PROPERTY ExecuteModelCode_Online : BOOL
GET
hResult := GetObjPara(16#00000008,sizeof(ExecuteModelCode_Online),adr(ExecuteModelCode_Online));
END_GET
SET
hResult := SetObjPara(16#00000008,sizeof(ExecuteModelCode_Online),adr(ExecuteModelCode_Online));
END_SET
END_PROPERTY

PROPERTY ExecuteModelCode_Startup : BOOL
GET
ExecuteModelCode_Startup := stInitData.ExecuteModelCode;
END_GET
SET
stInitData.ExecuteModelCode := ExecuteModelCode_Startup;
END_SET
END_PROPERTY

PROPERTY ExecutionSequence_Online : TctModuleExecutionSequenceType
GET
hResult := GetObjPara(16#00000001,sizeof(ExecutionSequence_Online),adr(ExecutionSequence_Online));
END_GET
SET
hResult := SetObjPara(16#00000001,sizeof(ExecutionSequence_Online),adr(ExecutionSequence_Online));
END_SET
END_PROPERTY

PROPERTY ExecutionSequence_Startup : TctModuleExecutionSequenceType
GET
ExecutionSequence_Startup := stInitData.ExecutionSequence;
END_GET
SET
stInitData.ExecutionSequence := ExecutionSequence_Startup;
END_SET
END_PROPERTY

METHOD FB_init : BOOL
VAR_INPUT
	/// if TRUE, the retain variables are initialized (warm start / cold start)
	bInitRetains: BOOL;
	/// if TRUE, the instance afterwards gets moved into the copy code (online change)
	bInCopyCode: BOOL;
	oid: OTCID;
END_VAR
VAR
	clsId: CLSID;
END_VAR

// initialize flags
bParametersVerified := false;
                    
// set module class id for compatibility check
clsId.Data1 := 16#4ef20903;
clsId.Data2 := 16#d648;
clsId.Data3 := 16#49c7;
clsId.Data4[0] := 16#a9;
clsId.Data4[1] := 16#06;
clsId.Data4[2] := 16#8c;
clsId.Data4[3] := 16#fc;
clsId.Data4[4] := 16#20;
clsId.Data4[5] := 16#50;
clsId.Data4[6] := 16#7f;
clsId.Data4[7] := 16#b3;

AssignClassId(clsId);
                    
// initialize InitData structure with default values              
stInitData.CallByHdr.indexGroup := 0;
stInitData.CallByHdr.indexOffset := 16#00000000;
stInitData.CallByHdr.cbData := SIZEOF(stInitData.CallBy);
stInitData.CallBy := TctModuleCallByType.Module;
stInitData.ExecutionSequenceHdr.indexGroup := 0;
stInitData.ExecutionSequenceHdr.indexOffset := 16#00000001;
stInitData.ExecutionSequenceHdr.cbData := SIZEOF(stInitData.ExecutionSequence);
stInitData.ExecutionSequence := TctModuleExecutionSequenceType.StateUpdateAfterOutputMapping;
stInitData.StepSizeHdr.indexGroup := 0;
stInitData.StepSizeHdr.indexOffset := 16#00000002;
stInitData.StepSizeHdr.cbData := SIZEOF(stInitData.StepSize);
stInitData.StepSize := TctStepSizeType.UseTaskCycleTime;
stInitData.ExecuteModelCodeHdr.indexGroup := 0;
stInitData.ExecuteModelCodeHdr.indexOffset := 16#00000008;
stInitData.ExecuteModelCodeHdr.cbData := SIZEOF(stInitData.ExecuteModelCode);
stInitData.ExecuteModelCode := 1;
stInitData.ModelParametersHdr.indexGroup := 0;
stInitData.ModelParametersHdr.indexOffset := 16#83000000;
stInitData.ModelParametersHdr.cbData := SIZEOF(stInitData.ModelParameters);
stInitData.ModelParameters.DiscreteFilter_NumCoef[0] := 1.25663706143591720e+01;
stInitData.ModelParameters.DiscreteFilter_NumCoef[1] := 1.25663706143591720e+01;
stInitData.ModelParameters.DiscreteFilter_DenCoef[0] := 2.01256637061435910e+03;
stInitData.ModelParameters.DiscreteFilter_DenCoef[1] := -1.98743362938564090e+03;
stInitData.ModelParameters.DiscreteFilter_InitialStates := 0.00000000000000000e+00;
stInitData.ModelParameters.DiscreteFilter1_NumCoef[0] := 1.25663706143591720e+01;
stInitData.ModelParameters.DiscreteFilter1_NumCoef[1] := 1.25663706143591720e+01;
stInitData.ModelParameters.DiscreteFilter1_DenCoef[0] := 2.01256637061435910e+03;
stInitData.ModelParameters.DiscreteFilter1_DenCoef[1] := -1.98743362938564090e+03;
stInitData.ModelParameters.DiscreteFilter1_InitialStates := 0.00000000000000000e+00;
stInitData.ModelParameters.DiscreteFilter2_NumCoef[0] := 1.25663706143591720e+01;
stInitData.ModelParameters.DiscreteFilter2_NumCoef[1] := 1.25663706143591720e+01;
stInitData.ModelParameters.DiscreteFilter2_DenCoef[0] := 2.01256637061435910e+03;
stInitData.ModelParameters.DiscreteFilter2_DenCoef[1] := -1.98743362938564090e+03;
stInitData.ModelParameters.DiscreteFilter2_InitialStates := 0.00000000000000000e+00;
stInitData.ModelParameters.DiscreteFilter3_NumCoef[0] := 1.25663706143591720e+01;
stInitData.ModelParameters.DiscreteFilter3_NumCoef[1] := 1.25663706143591720e+01;
stInitData.ModelParameters.DiscreteFilter3_DenCoef[0] := 2.01256637061435910e+03;
stInitData.ModelParameters.DiscreteFilter3_DenCoef[1] := -1.98743362938564090e+03;
stInitData.ModelParameters.DiscreteFilter3_InitialStates := 0.00000000000000000e+00;
stInitData.ModelParameters.DiscreteFilter4_NumCoef[0] := 1.25663706143591720e+01;
stInitData.ModelParameters.DiscreteFilter4_NumCoef[1] := 1.25663706143591720e+01;
stInitData.ModelParameters.DiscreteFilter4_DenCoef[0] := 2.01256637061435910e+03;
stInitData.ModelParameters.DiscreteFilter4_DenCoef[1] := -1.98743362938564090e+03;
stInitData.ModelParameters.DiscreteFilter4_InitialStates := 0.00000000000000000e+00;
stInitData.ModelParameters.DiscreteFilter5_NumCoef[0] := 1.25663706143591720e+01;
stInitData.ModelParameters.DiscreteFilter5_NumCoef[1] := 1.25663706143591720e+01;
stInitData.ModelParameters.DiscreteFilter5_DenCoef[0] := 2.01256637061435910e+03;
stInitData.ModelParameters.DiscreteFilter5_DenCoef[1] := -1.98743362938564090e+03;
stInitData.ModelParameters.DiscreteFilter5_InitialStates := 0.00000000000000000e+00;
stInitData.ModelParameters.DiscreteFilter6_NumCoef[0] := 1.25663706143591720e+01;
stInitData.ModelParameters.DiscreteFilter6_NumCoef[1] := 1.25663706143591720e+01;
stInitData.ModelParameters.DiscreteFilter6_DenCoef[0] := 2.01256637061435910e+03;
stInitData.ModelParameters.DiscreteFilter6_DenCoef[1] := -1.98743362938564090e+03;
stInitData.ModelParameters.DiscreteFilter6_InitialStates := 0.00000000000000000e+00;
stInitData.ModelParameters.DiscreteFilter7_NumCoef[0] := 1.25663706143591720e+01;
stInitData.ModelParameters.DiscreteFilter7_NumCoef[1] := 1.25663706143591720e+01;
stInitData.ModelParameters.DiscreteFilter7_DenCoef[0] := 2.01256637061435910e+03;
stInitData.ModelParameters.DiscreteFilter7_DenCoef[1] := -1.98743362938564090e+03;
stInitData.ModelParameters.DiscreteFilter7_InitialStates := 0.00000000000000000e+00;
stInitData.ModelParameters.DiscreteFilter8_NumCoef[0] := 1.25663706143591720e+01;
stInitData.ModelParameters.DiscreteFilter8_NumCoef[1] := 1.25663706143591720e+01;
stInitData.ModelParameters.DiscreteFilter8_DenCoef[0] := 2.01256637061435910e+03;
stInitData.ModelParameters.DiscreteFilter8_DenCoef[1] := -1.98743362938564090e+03;
stInitData.ModelParameters.DiscreteFilter8_InitialStates := 0.00000000000000000e+00;
stInitData.ModelParameters.DiscreteFilter9_NumCoef[0] := 1.25663706143591720e+01;
stInitData.ModelParameters.DiscreteFilter9_NumCoef[1] := 1.25663706143591720e+01;
stInitData.ModelParameters.DiscreteFilter9_DenCoef[0] := 2.01256637061435910e+03;
stInitData.ModelParameters.DiscreteFilter9_DenCoef[1] := -1.98743362938564090e+03;
stInitData.ModelParameters.DiscreteFilter9_InitialStates := 0.00000000000000000e+00;
stInitData.ModelParameters.DiscreteFilter10_NumCoef[0] := 1.25663706143591720e+01;
stInitData.ModelParameters.DiscreteFilter10_NumCoef[1] := 1.25663706143591720e+01;
stInitData.ModelParameters.DiscreteFilter10_DenCoef[0] := 2.01256637061435910e+03;
stInitData.ModelParameters.DiscreteFilter10_DenCoef[1] := -1.98743362938564090e+03;
stInitData.ModelParameters.DiscreteFilter10_InitialStates := 0.00000000000000000e+00;
stInitData.ModelParameters.DiscreteFilter11_NumCoef[0] := 1.25663706143591720e+01;
stInitData.ModelParameters.DiscreteFilter11_NumCoef[1] := 1.25663706143591720e+01;
stInitData.ModelParameters.DiscreteFilter11_DenCoef[0] := 2.01256637061435910e+03;
stInitData.ModelParameters.DiscreteFilter11_DenCoef[1] := -1.98743362938564090e+03;
stInitData.ModelParameters.DiscreteFilter11_InitialStates := 0.00000000000000000e+00;
stInitData.ModelParameters.DiscreteFilter12_NumCoef[0] := 1.25663706143591720e+01;
stInitData.ModelParameters.DiscreteFilter12_NumCoef[1] := 1.25663706143591720e+01;
stInitData.ModelParameters.DiscreteFilter12_DenCoef[0] := 2.01256637061435910e+03;
stInitData.ModelParameters.DiscreteFilter12_DenCoef[1] := -1.98743362938564090e+03;
stInitData.ModelParameters.DiscreteFilter12_InitialStates := 0.00000000000000000e+00;
stInitData.ModelParameters.DiscreteFilter13_NumCoef[0] := 1.25663706143591720e+01;
stInitData.ModelParameters.DiscreteFilter13_NumCoef[1] := 1.25663706143591720e+01;
stInitData.ModelParameters.DiscreteFilter13_DenCoef[0] := 2.01256637061435910e+03;
stInitData.ModelParameters.DiscreteFilter13_DenCoef[1] := -1.98743362938564090e+03;
stInitData.ModelParameters.DiscreteFilter13_InitialStates := 0.00000000000000000e+00;
stInitData.ModelParameters.DiscreteFilter14_NumCoef[0] := 1.25663706143591720e+01;
stInitData.ModelParameters.DiscreteFilter14_NumCoef[1] := 1.25663706143591720e+01;
stInitData.ModelParameters.DiscreteFilter14_DenCoef[0] := 2.01256637061435910e+03;
stInitData.ModelParameters.DiscreteFilter14_DenCoef[1] := -1.98743362938564090e+03;
stInitData.ModelParameters.DiscreteFilter14_InitialStates := 0.00000000000000000e+00;
stInitData.ModelParameters.DiscreteFilter15_NumCoef[0] := 1.25663706143591720e+01;
stInitData.ModelParameters.DiscreteFilter15_NumCoef[1] := 1.25663706143591720e+01;
stInitData.ModelParameters.DiscreteFilter15_DenCoef[0] := 2.01256637061435910e+03;
stInitData.ModelParameters.DiscreteFilter15_DenCoef[1] := -1.98743362938564090e+03;
stInitData.ModelParameters.DiscreteFilter15_InitialStates := 0.00000000000000000e+00;
stInitData.ModelParameters.DiscreteFilter16_NumCoef[0] := 1.25663706143591720e+01;
stInitData.ModelParameters.DiscreteFilter16_NumCoef[1] := 1.25663706143591720e+01;
stInitData.ModelParameters.DiscreteFilter16_DenCoef[0] := 2.01256637061435910e+03;
stInitData.ModelParameters.DiscreteFilter16_DenCoef[1] := -1.98743362938564090e+03;
stInitData.ModelParameters.DiscreteFilter16_InitialStates := 0.00000000000000000e+00;
stInitData.ModelParameters.DiscreteFilter17_NumCoef[0] := 1.25663706143591720e+01;
stInitData.ModelParameters.DiscreteFilter17_NumCoef[1] := 1.25663706143591720e+01;
stInitData.ModelParameters.DiscreteFilter17_DenCoef[0] := 2.01256637061435910e+03;
stInitData.ModelParameters.DiscreteFilter17_DenCoef[1] := -1.98743362938564090e+03;
stInitData.ModelParameters.DiscreteFilter17_InitialStates := 0.00000000000000000e+00;
stInitData.ContextInfoArr_0_TaskOidHdr.indexGroup := 0;
stInitData.ContextInfoArr_0_TaskOidHdr.indexOffset := 16#03002060;
stInitData.ContextInfoArr_0_TaskOidHdr.cbData := SIZEOF(stInitData.ContextInfoArr_0_TaskOid);
stInitData.ContextInfoArr_0_TaskPriorityHdr.indexGroup := 0;
stInitData.ContextInfoArr_0_TaskPriorityHdr.indexOffset := 16#03002070;
stInitData.ContextInfoArr_0_TaskPriorityHdr.cbData := SIZEOF(stInitData.ContextInfoArr_0_TaskPriority);
stInitData.ContextInfoArr_0_TaskCycleTimeNsHdr.indexGroup := 0;
stInitData.ContextInfoArr_0_TaskCycleTimeNsHdr.indexOffset := 16#03002080;
stInitData.ContextInfoArr_0_TaskCycleTimeNsHdr.cbData := SIZEOF(stInitData.ContextInfoArr_0_TaskCycleTimeNs);
stInitData.ContextInfoArr_0_TaskPortHdr.indexGroup := 0;
stInitData.ContextInfoArr_0_TaskPortHdr.indexOffset := 16#03002090;
stInitData.ContextInfoArr_0_TaskPortHdr.cbData := SIZEOF(stInitData.ContextInfoArr_0_TaskPort);
stInitData.ContextInfoArr_0_TaskSortOrderHdr.indexGroup := 0;
stInitData.ContextInfoArr_0_TaskSortOrderHdr.indexOffset := 16#030020b0;
stInitData.ContextInfoArr_0_TaskSortOrderHdr.cbData := SIZEOF(stInitData.ContextInfoArr_0_TaskSortOrder);
stInitData.Header.cbData := SIZEOF(stInitData)-SIZEOF(stInitData.Header);
stInitData.Header.uiElmCnt := 10;


// set pointer to InitData structure
SetInitDataInfo(ADR(stInitData));

// set DataArea information
SetDataAreaInfo(ADR(arrDataAreas),2);
arrDataAreas[1].nDataAreaId := 0;
arrDataAreas[1].nSize := SIZEOF(stInput);
arrDataAreas[1].pPlcVar := ADR(stInput);
arrDataAreas[1].pModuleProcImg := 0;
arrDataAreas[1].eDataAreaType := E_TcMatSimDataAreaType.InputDst;
arrDataAreas[2].nDataAreaId := 1;
arrDataAreas[2].nSize := SIZEOF(stOutput);
arrDataAreas[2].pPlcVar := ADR(stOutput);
arrDataAreas[2].pModuleProcImg := 0;
arrDataAreas[2].eDataAreaType := E_TcMatSimDataAreaType.OutputSrc;


// initialize basic interface pointers and return
FB_init := SUCCEEDED(Init(oid));
END_METHOD

PROPERTY InitData : ST_Filter_Current_Hexapod_Robot_InitData
GET
InitData := stInitData;
END_GET
SET
stInitData := InitData;
END_SET
END_PROPERTY

PROPERTY Input_Online : ExtU_Filter_Current_Hexapod_R_T
GET
hResult := GetObjPara(16#80000000,sizeof(Input_Online),adr(Input_Online));
END_GET
SET
hResult := SetObjPara(16#80000000,sizeof(Input_Online),adr(Input_Online));
END_SET
END_PROPERTY

{attribute 'object_name' := 'Internal_SetObjState'}
METHOD PROTECTED Internal_SetObjState
VAR_INPUT
	hr: REFERENCE TO HRESULT;
	nextState: TCOM_STATE;
END_VAR

// update pointer to InitData structure
SetInitDataInfo(ADR(stInitData));
// call base method
SUPER^.Internal_SetObjState(hr,nextState);
END_METHOD

PROPERTY MdlInitialized_Online : BOOL
GET
hResult := GetObjPara(16#00000003,sizeof(MdlInitialized_Online),adr(MdlInitialized_Online));
END_GET
SET
hResult := SetObjPara(16#00000003,sizeof(MdlInitialized_Online),adr(MdlInitialized_Online));
END_SET
END_PROPERTY

PROPERTY ModelParameters_Online : P_Filter_Current_Hexapod_Robo_T
GET
hResult := GetObjPara(16#83000000,sizeof(ModelParameters_Online),adr(ModelParameters_Online));
END_GET
SET
hResult := SetObjPara(16#83000000,sizeof(ModelParameters_Online),adr(ModelParameters_Online));
END_SET
END_PROPERTY

PROPERTY ModelParameters_Startup : P_Filter_Current_Hexapod_Robo_T
GET
ModelParameters_Startup := stInitData.ModelParameters;
END_GET
SET
stInitData.ModelParameters := ModelParameters_Startup;
END_SET
END_PROPERTY

PROPERTY ModuleBuildInfo_Online : TctModuleBuildInfoType
GET
hResult := GetObjPara(16#00000007,sizeof(ModuleBuildInfo_Online),adr(ModuleBuildInfo_Online));
END_GET
SET
hResult := SetObjPara(16#00000007,sizeof(ModuleBuildInfo_Online),adr(ModuleBuildInfo_Online));
END_SET
END_PROPERTY

PROPERTY ModuleInfo_Online : TctModuleInfoType
GET
hResult := GetObjPara(16#00000006,sizeof(ModuleInfo_Online),adr(ModuleInfo_Online));
END_GET
SET
hResult := SetObjPara(16#00000006,sizeof(ModuleInfo_Online),adr(ModuleInfo_Online));
END_SET
END_PROPERTY

{attribute 'object_name' := 'SaveOnlineParametersForInit'}
METHOD SaveOnlineParametersForInit : HRESULT
VAR
	idx: UINT;
	pInitElemHdr: POINTER TO TComInitDataElmHdr;
	pData: PVOID;
	nData: UDINT;
END_VAR
VAR CONSTANT
	nInitDataAlignment: UDINT := 4;
END_VAR

// update pointer to InitData structure
SetInitDataInfo(ADR(stInitData));
// call base method
SaveOnlineParametersForInit := SUPER^.SaveOnlineParametersForInit();
END_METHOD

PROPERTY SimulinkTime_Online : LREAL
GET
hResult := GetObjPara(16#00000005,sizeof(SimulinkTime_Online),adr(SimulinkTime_Online));
END_GET
SET
hResult := SetObjPara(16#00000005,sizeof(SimulinkTime_Online),adr(SimulinkTime_Online));
END_SET
END_PROPERTY

PROPERTY StepSize_Online : TctStepSizeType
GET
hResult := GetObjPara(16#00000002,sizeof(StepSize_Online),adr(StepSize_Online));
END_GET
SET
hResult := SetObjPara(16#00000002,sizeof(StepSize_Online),adr(StepSize_Online));
END_SET
END_PROPERTY

PROPERTY StepSize_Startup : TctStepSizeType
GET
StepSize_Startup := stInitData.StepSize;
END_GET
SET
stInitData.StepSize := StepSize_Startup;
END_SET
END_PROPERTY

{attribute 'object_name' := 'VerifyParameters'}
METHOD PRIVATE VerifyParameters : HRESULT
VAR
	moduleCallByParam: TctModuleCallByType;
END_VAR

IF (bParametersVerified) THEN
  VerifyParameters := Tc2_System.E_HRESULTAdsErr.HRESULT_ADS_NOERROR;
ELSE
  VerifyParameters := GetObjPara(stInitData.CallByHdr.indexOffset,SIZEOF(moduleCallByParam),ADR(moduleCallByParam));
  
  // check the "CallBy" parameter to be set to "Module"
  IF (SUCCEEDED(VerifyParameters) AND (moduleCallByParam <> TctModuleCallByType.Module)) THEN
      VerifyParameters := Tc2_System.E_HRESULTAdsErr.INVALIDPARM;
  END_IF
  
  // set the parameters verified flag
  bParametersVerified := SUCCEEDED(VerifyParameters);
END_IF
END_METHOD

END_FUNCTION_BLOCK

// ---- DUTs/Touch_Signal_Detection/FB_Tough_Signal_Detection_Simple.TcPOU
{attribute 'TcDependOnClassFactory' := 'Tough_Signal_Detection_Simple'}
FUNCTION_BLOCK FB_Tough_Signal_Detection_Simple EXTENDS FB_TcMatSimObject
VAR_INPUT
	stInput: ST_Tough_Signal_Detection_Simple_Input;
END_VAR
VAR_OUTPUT
	stOutput: ST_Tough_Signal_Detection_Simple_Output;
END_VAR
VAR
	stInitData: ST_Tough_Signal_Detection_Simple_InitData;
	arrDataAreas: ARRAY[1..2] OF ST_TcMatSimObjectDataAreaInfo;
	bParametersVerified: BOOL;
END_VAR

PROPERTY CallBy_Online : TctModuleCallByType
GET
hResult := GetObjPara(16#00000000,sizeof(CallBy_Online),adr(CallBy_Online));
END_GET
SET
hResult := SetObjPara(16#00000000,sizeof(CallBy_Online),adr(CallBy_Online));
END_SET
END_PROPERTY

PROPERTY CallBy_Startup : TctModuleCallByType
GET
CallBy_Startup := stInitData.CallBy;
END_GET
SET
stInitData.CallBy := CallBy_Startup;
END_SET
END_PROPERTY

PROPERTY ContextInfoArr_0_TaskCycleTimeNs_Online : UDINT
GET
hResult := GetObjPara(16#03002080,sizeof(ContextInfoArr_0_TaskCycleTimeNs_Online),adr(ContextInfoArr_0_TaskCycleTimeNs_Online));
END_GET
SET
hResult := SetObjPara(16#03002080,sizeof(ContextInfoArr_0_TaskCycleTimeNs_Online),adr(ContextInfoArr_0_TaskCycleTimeNs_Online));
END_SET
END_PROPERTY

PROPERTY ContextInfoArr_0_TaskCycleTimeNs_Startup : UDINT
GET
ContextInfoArr_0_TaskCycleTimeNs_Startup := stInitData.ContextInfoArr_0_TaskCycleTimeNs;
END_GET
SET
stInitData.ContextInfoArr_0_TaskCycleTimeNs := ContextInfoArr_0_TaskCycleTimeNs_Startup;
END_SET
END_PROPERTY

PROPERTY ContextInfoArr_0_TaskOid_Online : OTCID
GET
hResult := GetObjPara(16#03002060,sizeof(ContextInfoArr_0_TaskOid_Online),adr(ContextInfoArr_0_TaskOid_Online));
END_GET
SET
hResult := SetObjPara(16#03002060,sizeof(ContextInfoArr_0_TaskOid_Online),adr(ContextInfoArr_0_TaskOid_Online));
END_SET
END_PROPERTY

PROPERTY ContextInfoArr_0_TaskOid_Startup : OTCID
GET
ContextInfoArr_0_TaskOid_Startup := stInitData.ContextInfoArr_0_TaskOid;
END_GET
SET
stInitData.ContextInfoArr_0_TaskOid := ContextInfoArr_0_TaskOid_Startup;
END_SET
END_PROPERTY

PROPERTY ContextInfoArr_0_TaskPort_Online : UINT
GET
hResult := GetObjPara(16#03002090,sizeof(ContextInfoArr_0_TaskPort_Online),adr(ContextInfoArr_0_TaskPort_Online));
END_GET
SET
hResult := SetObjPara(16#03002090,sizeof(ContextInfoArr_0_TaskPort_Online),adr(ContextInfoArr_0_TaskPort_Online));
END_SET
END_PROPERTY

PROPERTY ContextInfoArr_0_TaskPort_Startup : UINT
GET
ContextInfoArr_0_TaskPort_Startup := stInitData.ContextInfoArr_0_TaskPort;
END_GET
SET
stInitData.ContextInfoArr_0_TaskPort := ContextInfoArr_0_TaskPort_Startup;
END_SET
END_PROPERTY

PROPERTY ContextInfoArr_0_TaskPriority_Online : UDINT
GET
hResult := GetObjPara(16#03002070,sizeof(ContextInfoArr_0_TaskPriority_Online),adr(ContextInfoArr_0_TaskPriority_Online));
END_GET
SET
hResult := SetObjPara(16#03002070,sizeof(ContextInfoArr_0_TaskPriority_Online),adr(ContextInfoArr_0_TaskPriority_Online));
END_SET
END_PROPERTY

PROPERTY ContextInfoArr_0_TaskPriority_Startup : UDINT
GET
ContextInfoArr_0_TaskPriority_Startup := stInitData.ContextInfoArr_0_TaskPriority;
END_GET
SET
stInitData.ContextInfoArr_0_TaskPriority := ContextInfoArr_0_TaskPriority_Startup;
END_SET
END_PROPERTY

PROPERTY ContextInfoArr_0_TaskSortOrder_Online : UDINT
GET
hResult := GetObjPara(16#030020b0,sizeof(ContextInfoArr_0_TaskSortOrder_Online),adr(ContextInfoArr_0_TaskSortOrder_Online));
END_GET
SET
hResult := SetObjPara(16#030020b0,sizeof(ContextInfoArr_0_TaskSortOrder_Online),adr(ContextInfoArr_0_TaskSortOrder_Online));
END_SET
END_PROPERTY

PROPERTY ContextInfoArr_0_TaskSortOrder_Startup : UDINT
GET
ContextInfoArr_0_TaskSortOrder_Startup := stInitData.ContextInfoArr_0_TaskSortOrder;
END_GET
SET
stInitData.ContextInfoArr_0_TaskSortOrder := ContextInfoArr_0_TaskSortOrder_Startup;
END_SET
END_PROPERTY

PROPERTY CycleUpdateExecuted_Online : BOOL
GET
hResult := GetObjPara(16#00000004,sizeof(CycleUpdateExecuted_Online),adr(CycleUpdateExecuted_Online));
END_GET
SET
hResult := SetObjPara(16#00000004,sizeof(CycleUpdateExecuted_Online),adr(CycleUpdateExecuted_Online));
END_SET
END_PROPERTY

METHOD Execute : HRESULT

IF (SUCCEEDED(hResult)) THEN
  hResult := VerifyParameters();
END_IF

	// update DataArea information
SetDataAreaInfo(ADR(arrDataAreas),2);
	
	// call base method
Execute := SUPER^.Execute();
END_METHOD

PROPERTY ExecuteModelCode_Online : BOOL
GET
hResult := GetObjPara(16#00000008,sizeof(ExecuteModelCode_Online),adr(ExecuteModelCode_Online));
END_GET
SET
hResult := SetObjPara(16#00000008,sizeof(ExecuteModelCode_Online),adr(ExecuteModelCode_Online));
END_SET
END_PROPERTY

PROPERTY ExecuteModelCode_Startup : BOOL
GET
ExecuteModelCode_Startup := stInitData.ExecuteModelCode;
END_GET
SET
stInitData.ExecuteModelCode := ExecuteModelCode_Startup;
END_SET
END_PROPERTY

PROPERTY ExecutionSequence_Online : TctModuleExecutionSequenceType
GET
hResult := GetObjPara(16#00000001,sizeof(ExecutionSequence_Online),adr(ExecutionSequence_Online));
END_GET
SET
hResult := SetObjPara(16#00000001,sizeof(ExecutionSequence_Online),adr(ExecutionSequence_Online));
END_SET
END_PROPERTY

PROPERTY ExecutionSequence_Startup : TctModuleExecutionSequenceType
GET
ExecutionSequence_Startup := stInitData.ExecutionSequence;
END_GET
SET
stInitData.ExecutionSequence := ExecutionSequence_Startup;
END_SET
END_PROPERTY

METHOD FB_init : BOOL
VAR_INPUT
	/// if TRUE, the retain variables are initialized (warm start / cold start)
	bInitRetains: BOOL;
	/// if TRUE, the instance afterwards gets moved into the copy code (online change)
	bInCopyCode: BOOL;
	oid: OTCID;
END_VAR
VAR
	clsId: CLSID;
END_VAR

// initialize flags
bParametersVerified := false;
                    
// set module class id for compatibility check
clsId.Data1 := 16#edbb4036;
clsId.Data2 := 16#240d;
clsId.Data3 := 16#4fd3;
clsId.Data4[0] := 16#9b;
clsId.Data4[1] := 16#53;
clsId.Data4[2] := 16#34;
clsId.Data4[3] := 16#bf;
clsId.Data4[4] := 16#ff;
clsId.Data4[5] := 16#27;
clsId.Data4[6] := 16#d6;
clsId.Data4[7] := 16#ef;

AssignClassId(clsId);
                    
// initialize InitData structure with default values              
stInitData.CallByHdr.indexGroup := 0;
stInitData.CallByHdr.indexOffset := 16#00000000;
stInitData.CallByHdr.cbData := SIZEOF(stInitData.CallBy);
stInitData.CallBy := TctModuleCallByType.Module;
stInitData.ExecutionSequenceHdr.indexGroup := 0;
stInitData.ExecutionSequenceHdr.indexOffset := 16#00000001;
stInitData.ExecutionSequenceHdr.cbData := SIZEOF(stInitData.ExecutionSequence);
stInitData.ExecutionSequence := TctModuleExecutionSequenceType.StateUpdateAfterOutputMapping;
stInitData.StepSizeHdr.indexGroup := 0;
stInitData.StepSizeHdr.indexOffset := 16#00000002;
stInitData.StepSizeHdr.cbData := SIZEOF(stInitData.StepSize);
stInitData.StepSize := TctStepSizeType.UseTaskCycleTime;
stInitData.ExecuteModelCodeHdr.indexGroup := 0;
stInitData.ExecuteModelCodeHdr.indexOffset := 16#00000008;
stInitData.ExecuteModelCodeHdr.cbData := SIZEOF(stInitData.ExecuteModelCode);
stInitData.ExecuteModelCode := 1;
stInitData.ModelParametersHdr.indexGroup := 0;
stInitData.ModelParametersHdr.indexOffset := 16#83000000;
stInitData.ModelParametersHdr.cbData := SIZEOF(stInitData.ModelParameters);
stInitData.ModelParameters.VariableTimeDelay_MaxDelay := 1.00000000000000000e+00;
stInitData.ModelParameters.VariableTimeDelay_InitOutput := 0.00000000000000000e+00;
stInitData.ModelParameters.VariableTimeDelay1_MaxDelay := 1.00000000000000000e+00;
stInitData.ModelParameters.VariableTimeDelay1_InitOutput := 0.00000000000000000e+00;
stInitData.ModelParameters.VariableTimeDelay2_MaxDelay := 1.00000000000000000e+00;
stInitData.ModelParameters.VariableTimeDelay2_InitOutput := 0.00000000000000000e+00;
stInitData.ModelParameters.VariableTimeDelay3_MaxDelay := 1.00000000000000000e+00;
stInitData.ModelParameters.VariableTimeDelay3_InitOutput := 0.00000000000000000e+00;
stInitData.ModelParameters.VariableTimeDelay4_MaxDelay := 1.00000000000000000e+00;
stInitData.ModelParameters.VariableTimeDelay4_InitOutput := 0.00000000000000000e+00;
stInitData.ModelParameters.VariableTimeDelay5_MaxDelay := 1.00000000000000000e+00;
stInitData.ModelParameters.VariableTimeDelay5_InitOutput := 0.00000000000000000e+00;
stInitData.ModelParameters.VariableTimeDelay6_MaxDelay := 1.00000000000000000e+00;
stInitData.ModelParameters.VariableTimeDelay6_InitOutput := 0.00000000000000000e+00;
stInitData.ModelParameters.VariableTimeDelay7_MaxDelay := 1.00000000000000000e+00;
stInitData.ModelParameters.VariableTimeDelay7_InitOutput := 0.00000000000000000e+00;
stInitData.ModelParameters.VariableTimeDelay8_MaxDelay := 1.00000000000000000e+00;
stInitData.ModelParameters.VariableTimeDelay8_InitOutput := 0.00000000000000000e+00;
stInitData.ModelParameters.VariableTimeDelay9_MaxDelay := 1.00000000000000000e+00;
stInitData.ModelParameters.VariableTimeDelay9_InitOutput := 0.00000000000000000e+00;
stInitData.ModelParameters.VariableTimeDelay10_MaxDelay := 1.00000000000000000e+00;
stInitData.ModelParameters.VariableTimeDelay10_InitOutput := 0.00000000000000000e+00;
stInitData.ModelParameters.VariableTimeDelay11_MaxDelay := 1.00000000000000000e+00;
stInitData.ModelParameters.VariableTimeDelay11_InitOutput := 0.00000000000000000e+00;
stInitData.ModelParameters.VariableTimeDelay12_MaxDelay := 1.00000000000000000e+00;
stInitData.ModelParameters.VariableTimeDelay12_InitOutput := 0.00000000000000000e+00;
stInitData.ModelParameters.VariableTimeDelay13_MaxDelay := 1.00000000000000000e+00;
stInitData.ModelParameters.VariableTimeDelay13_InitOutput := 0.00000000000000000e+00;
stInitData.ModelParameters.VariableTimeDelay14_MaxDelay := 1.00000000000000000e+00;
stInitData.ModelParameters.VariableTimeDelay14_InitOutput := 0.00000000000000000e+00;
stInitData.ModelParameters.VariableTimeDelay15_MaxDelay := 1.00000000000000000e+00;
stInitData.ModelParameters.VariableTimeDelay15_InitOutput := 0.00000000000000000e+00;
stInitData.ModelParameters.VariableTimeDelay16_MaxDelay := 1.00000000000000000e+00;
stInitData.ModelParameters.VariableTimeDelay16_InitOutput := 0.00000000000000000e+00;
stInitData.ModelParameters.VariableTimeDelay17_MaxDelay := 1.00000000000000000e+00;
stInitData.ModelParameters.VariableTimeDelay17_InitOutput := 0.00000000000000000e+00;
stInitData.ModelParameters.DataStoreMemory5_InitialValue[0] := 1.00000000000000000e+00;
stInitData.ModelParameters.DataStoreMemory5_InitialValue[1] := 3.00000000000000000e+00;
stInitData.ModelParameters.DataStoreMemory5_InitialValue[2] := 5.00000000000000000e+00;
stInitData.ModelParameters.DataStoreMemory6_InitialValue[0] := 2.00000000000000000e+00;
stInitData.ModelParameters.DataStoreMemory6_InitialValue[1] := 4.00000000000000000e+00;
stInitData.ModelParameters.DataStoreMemory6_InitialValue[2] := 6.00000000000000000e+00;
stInitData.ModelParameters.DataStoreMemory4_InitialValue[0] := 1;
stInitData.ModelParameters.DataStoreMemory4_InitialValue[1] := 0;
stInitData.ModelParameters.DataStoreMemory4_InitialValue[2] := 1;
stInitData.ModelParameters.DataStoreMemory4_InitialValue[3] := 0;
stInitData.ModelParameters.DataStoreMemory4_InitialValue[4] := 1;
stInitData.ModelParameters.DataStoreMemory4_InitialValue[5] := 0;
stInitData.ContextInfoArr_0_TaskOidHdr.indexGroup := 0;
stInitData.ContextInfoArr_0_TaskOidHdr.indexOffset := 16#03002060;
stInitData.ContextInfoArr_0_TaskOidHdr.cbData := SIZEOF(stInitData.ContextInfoArr_0_TaskOid);
stInitData.ContextInfoArr_0_TaskPriorityHdr.indexGroup := 0;
stInitData.ContextInfoArr_0_TaskPriorityHdr.indexOffset := 16#03002070;
stInitData.ContextInfoArr_0_TaskPriorityHdr.cbData := SIZEOF(stInitData.ContextInfoArr_0_TaskPriority);
stInitData.ContextInfoArr_0_TaskCycleTimeNsHdr.indexGroup := 0;
stInitData.ContextInfoArr_0_TaskCycleTimeNsHdr.indexOffset := 16#03002080;
stInitData.ContextInfoArr_0_TaskCycleTimeNsHdr.cbData := SIZEOF(stInitData.ContextInfoArr_0_TaskCycleTimeNs);
stInitData.ContextInfoArr_0_TaskPortHdr.indexGroup := 0;
stInitData.ContextInfoArr_0_TaskPortHdr.indexOffset := 16#03002090;
stInitData.ContextInfoArr_0_TaskPortHdr.cbData := SIZEOF(stInitData.ContextInfoArr_0_TaskPort);
stInitData.ContextInfoArr_0_TaskSortOrderHdr.indexGroup := 0;
stInitData.ContextInfoArr_0_TaskSortOrderHdr.indexOffset := 16#030020b0;
stInitData.ContextInfoArr_0_TaskSortOrderHdr.cbData := SIZEOF(stInitData.ContextInfoArr_0_TaskSortOrder);
stInitData.Header.cbData := SIZEOF(stInitData)-SIZEOF(stInitData.Header);
stInitData.Header.uiElmCnt := 10;


// set pointer to InitData structure
SetInitDataInfo(ADR(stInitData));

// set DataArea information
SetDataAreaInfo(ADR(arrDataAreas),2);
arrDataAreas[1].nDataAreaId := 0;
arrDataAreas[1].nSize := SIZEOF(stInput);
arrDataAreas[1].pPlcVar := ADR(stInput);
arrDataAreas[1].pModuleProcImg := 0;
arrDataAreas[1].eDataAreaType := E_TcMatSimDataAreaType.InputDst;
arrDataAreas[2].nDataAreaId := 1;
arrDataAreas[2].nSize := SIZEOF(stOutput);
arrDataAreas[2].pPlcVar := ADR(stOutput);
arrDataAreas[2].pModuleProcImg := 0;
arrDataAreas[2].eDataAreaType := E_TcMatSimDataAreaType.OutputSrc;


// initialize basic interface pointers and return
FB_init := SUCCEEDED(Init(oid));
END_METHOD

PROPERTY InitData : ST_Tough_Signal_Detection_Simple_InitData
GET
InitData := stInitData;
END_GET
SET
stInitData := InitData;
END_SET
END_PROPERTY

PROPERTY Input_Online : ExtU_Touch_Signal_Detection_S_T
GET
hResult := GetObjPara(16#80000000,sizeof(Input_Online),adr(Input_Online));
END_GET
SET
hResult := SetObjPara(16#80000000,sizeof(Input_Online),adr(Input_Online));
END_SET
END_PROPERTY

{attribute 'object_name' := 'Internal_SetObjState'}
METHOD PROTECTED Internal_SetObjState
VAR_INPUT
	hr: REFERENCE TO HRESULT;
	nextState: TCOM_STATE;
END_VAR

// update pointer to InitData structure
SetInitDataInfo(ADR(stInitData));
// call base method
SUPER^.Internal_SetObjState(hr,nextState);
END_METHOD

PROPERTY MdlInitialized_Online : BOOL
GET
hResult := GetObjPara(16#00000003,sizeof(MdlInitialized_Online),adr(MdlInitialized_Online));
END_GET
SET
hResult := SetObjPara(16#00000003,sizeof(MdlInitialized_Online),adr(MdlInitialized_Online));
END_SET
END_PROPERTY

PROPERTY ModelParameters_Online : P_Touch_Signal_Detection_Simp_T
GET
hResult := GetObjPara(16#83000000,sizeof(ModelParameters_Online),adr(ModelParameters_Online));
END_GET
SET
hResult := SetObjPara(16#83000000,sizeof(ModelParameters_Online),adr(ModelParameters_Online));
END_SET
END_PROPERTY

PROPERTY ModelParameters_Startup : P_Touch_Signal_Detection_Simp_T
GET
ModelParameters_Startup := stInitData.ModelParameters;
END_GET
SET
stInitData.ModelParameters := ModelParameters_Startup;
END_SET
END_PROPERTY

PROPERTY ModuleBuildInfo_Online : TctModuleBuildInfoType
GET
hResult := GetObjPara(16#00000007,sizeof(ModuleBuildInfo_Online),adr(ModuleBuildInfo_Online));
END_GET
SET
hResult := SetObjPara(16#00000007,sizeof(ModuleBuildInfo_Online),adr(ModuleBuildInfo_Online));
END_SET
END_PROPERTY

PROPERTY ModuleInfo_Online : TctModuleInfoType
GET
hResult := GetObjPara(16#00000006,sizeof(ModuleInfo_Online),adr(ModuleInfo_Online));
END_GET
SET
hResult := SetObjPara(16#00000006,sizeof(ModuleInfo_Online),adr(ModuleInfo_Online));
END_SET
END_PROPERTY

{attribute 'object_name' := 'SaveOnlineParametersForInit'}
METHOD SaveOnlineParametersForInit : HRESULT
VAR
	idx: UINT;
	pInitElemHdr: POINTER TO TComInitDataElmHdr;
	pData: PVOID;
	nData: UDINT;
END_VAR
VAR CONSTANT
	nInitDataAlignment: UDINT := 4;
END_VAR

// update pointer to InitData structure
SetInitDataInfo(ADR(stInitData));
// call base method
SaveOnlineParametersForInit := SUPER^.SaveOnlineParametersForInit();
END_METHOD

PROPERTY SimulinkTime_Online : LREAL
GET
hResult := GetObjPara(16#00000005,sizeof(SimulinkTime_Online),adr(SimulinkTime_Online));
END_GET
SET
hResult := SetObjPara(16#00000005,sizeof(SimulinkTime_Online),adr(SimulinkTime_Online));
END_SET
END_PROPERTY

PROPERTY StepSize_Online : TctStepSizeType
GET
hResult := GetObjPara(16#00000002,sizeof(StepSize_Online),adr(StepSize_Online));
END_GET
SET
hResult := SetObjPara(16#00000002,sizeof(StepSize_Online),adr(StepSize_Online));
END_SET
END_PROPERTY

PROPERTY StepSize_Startup : TctStepSizeType
GET
StepSize_Startup := stInitData.StepSize;
END_GET
SET
stInitData.StepSize := StepSize_Startup;
END_SET
END_PROPERTY

{attribute 'object_name' := 'VerifyParameters'}
METHOD PRIVATE VerifyParameters : HRESULT
VAR
	moduleCallByParam: TctModuleCallByType;
END_VAR

IF (bParametersVerified) THEN
  VerifyParameters := Tc2_System.E_HRESULTAdsErr.HRESULT_ADS_NOERROR;
ELSE
  VerifyParameters := GetObjPara(stInitData.CallByHdr.indexOffset,SIZEOF(moduleCallByParam),ADR(moduleCallByParam));
  
  // check the "CallBy" parameter to be set to "Module"
  IF (SUCCEEDED(VerifyParameters) AND (moduleCallByParam <> TctModuleCallByType.Module)) THEN
      VerifyParameters := Tc2_System.E_HRESULTAdsErr.INVALIDPARM;
  END_IF
  
  // set the parameters verified flag
  bParametersVerified := SUCCEEDED(VerifyParameters);
END_IF
END_METHOD

END_FUNCTION_BLOCK

// ---- POUs/Walking_Welding_Robot_Control.TcPOU
PROGRAM Walking_Welding_Robot_Control
VAR_INPUT
	// ====== 整体界面激活 ======
	Walking_Welding_Robot_Joint_Control	: BOOL;				// 允许对界面进行操作,对应UI中的Enable_All_Buttons
	
	// ====== 模块使能信号 ======
	Walking_Welding_Robot_Power 		: BOOL;				// [24电机上电]
	Walking_Welding_Robot_Home_Execute	: BOOL;				// [找零使能]
	Walking_Welding_Robot_Moving_Execute: BOOL;				// [运动使能]
	
	// ====== 控制类型选择 ======
	User_Moving_Control					: BOOL;				// 用户输入目标位置进行运动
	Auto_Moving_Control					: BOOL;				// 机器人自主根据Walking_Robot_Movement的默认参数进行运动
END_VAR

VAR
	// ===================控制信号输入=============
	// 六足运动位置定义(按潘阳坐标系) - 用户操作控制
		// 用户指定目标位置
	Robot_Walking_Z						: LREAL := 1.00;	// 用户指定运动 : Z方向目标位置
	Robot_Walking_X						: LREAL := 0.40;	// 用户指定运动 : X方向目标位置
	Robot_Walking_alpha					: LREAL := pi/12;	// 用户指定运动 : 绕Y轴旋转角度
	Robot_Walking_Velocity				: LREAL := 0.03;	// 用户指定运动 : 机器人运动速度默认0.03m/s
		// 机器人各方向运动速度
	Robot_Walking_Vx					: LREAL;			// X方向运动速度
	Robot_Walking_Vz					: LREAL;			// Z方向运动速度
	Robot_Walking_Va					: LREAL;			// Y方向转动速度
		// 机器人从当前位置运动到目标位置所需时间
	Robot_Walking_t						: LREAL;			// 运动总时间
END_VAR


Logic_Control();			// 逻辑控制程序

Input_Calculate();			// 用户输入参数计算

ACTION Input_Calculate:



// 用户指定目标位置,以当前位置为[0,0,0,0,0,0],按照机器人进行匀速运动,计算三个方向的速度
	// 沿X方向移动的速度分量 Vx = V * sin(theta)
Robot_Walking_Vx 	:= Robot_Walking_Velocity * SIN(ATAN(Robot_Walking_X/Robot_Walking_Z));
	// 沿Z方向移动的速度分量 Vz = V * cos(theta)
Robot_Walking_Vz 	:= Robot_Walking_Velocity * COS(ATAN(Robot_Walking_X/Robot_Walking_Z));
	// 机器人运动的总时间 t = Z / Vz
Robot_Walking_t		:= Robot_Walking_Z / Robot_Walking_Vz;	
	// 沿Y方向转动的速度分量 Va = alpha / t
Robot_Walking_Va	:= Robot_Walking_alpha / Robot_Walking_t;


// Simulink里的模型是以最开始的位置为全局坐标系,走到目标位置后
// 再想走一段的话重新给Vx,Vz,Va会发生什么呢？  

// 如果此时将Simulink模型的输入时间改为t=0会发生什么
END_ACTION

ACTION Logic_Control:
// ************************整体移动焊接机器人控制逻辑***********************

//  激活整个模块后,允许使用界面上的按钮进行操作,这样才能进行整体上电、找零、运动
IF Walking_Welding_Robot_Joint_control THEN
	// 上电、找零、运动三者逻辑
		// 未上电,不能找零和运动
	IF NOT Walking_Welding_Robot_Power THEN
		Walking_Welding_Robot_Home_Execute 	:= FALSE;
		Walking_Welding_Robot_Moving_Execute:= FALSE;
	END_IF
		// 找零时,不能运动
	IF Walking_Welding_Robot_Home_Execute THEN
		Walking_Welding_Robot_Moving_Execute:= FALSE;
	END_IF
		// 运动时,不能找零
	IF Walking_Welding_Robot_Moving_Execute THEN
		Walking_Welding_Robot_Home_Execute 	:= FALSE;
	END_IF	

	// 上电逻辑
		// [24电机上电]开启,则通过对应的控制PRG直接将所有电机整体上电
	IF Walking_Welding_Robot_Power THEN
		Walking_Robot_Control.Power_Execute 	:= TRUE;
		Walking_Robot_Control.Robot_Power		:= TRUE;
		Welding_Arm_Control.Power_Execute 		:= TRUE;
		Welding_Arm_Control.Welding_Arm_Power 	:= TRUE;
		// [24电机上电]关闭,通过对应的控制PRG直接将所有电机整体断电
	ELSIF NOT Walking_Welding_Robot_Power THEN
		Walking_Robot_Control.Power_Execute 	:= FALSE;
		Walking_Robot_Control.Robot_Power		:= FALSE;
		Welding_Arm_Control.Power_Execute 		:= FALSE;	
		Welding_Arm_Control.Welding_Arm_Power	:= FALSE;
	END_IF
		
	// 找零逻辑
		// [找零使能],则允许用户对焊接臂/步行机器人分别进行整体找零
		// 但仅仅是允许,找零动作的发生还需要用户通过界面上的按钮进行操作
	IF Walking_Welding_Robot_Home_Execute THEN
		Walking_Robot_Control.Home_Execute 		:= TRUE;	// 六足找零使能开启
		Walking_Robot_Control.Robot_Home_Set	:= TRUE;	// 六足单组退找零使能开启
		Welding_Arm_Control.Home_Execute 		:= TRUE;	// 焊接臂找零使能开启
	ELSIF NOT Walking_Welding_Robot_Home_Execute THEN
		Walking_Robot_Control.Home_Execute 		:= FALSE;
		Walking_Robot_Control.Robot_Home_Set	:= FALSE;
		Welding_Arm_Control.Home_Execute 		:= FALSE;
	END_IF
	
	// 两种控制方式互斥
	IF User_Moving_Control THEN
		Auto_Moving_Control := FALSE;
	END_IF
	IF Auto_Moving_Control THEN
		User_Moving_Control := FALSE;
	END_IF
	
	// 运动控制逻辑
	IF Walking_Welding_Robot_Moving_Execute THEN
		// [运动使能],则允许用户对焊接臂/步行机器人分别进行运动控制,即两者外部发生使能
		Walking_Robot_Movement.ExSetPoint_Execute 		:= TRUE;
		Welding_Arm_Movement.ExSetPoint_Execute 		:= TRUE;

		IF User_Moving_Control THEN
			Walking_Robot_Movement.ExtSetPointEnable	:= TRUE;
			Walking_Robot_Movement.ExtSetPointDisable	:= FALSE;
		ELSIF NOT User_Moving_Control THEN
			Walking_Robot_Movement.ExtSetPointEnable	:= FALSE;
			Walking_Robot_Movement.ExtSetPointDisable	:= TRUE;
		END_IF
		
	ELSIF NOT Walking_Welding_Robot_Moving_Execute THEN
		// [运动使能]关闭,不允许控制,且外部发生使能关闭
		Auto_Moving_Control := FALSE;
		User_Moving_Control := FALSE;
		Walking_Robot_Movement.ExSetPoint_Execute 	:= FALSE;
		Welding_Arm_Movement.ExSetPoint_Execute 	:= FALSE;
	END_IF
	
		// 用户自定义行走,走到目标位置后停止
	IF User_Moving_Control THEN
		// 到达目标位置附近后停止
		
		IF (Robot_Walking_Z-Walking_Robot_Movement.Act_Slice[3])< 0.15 AND (Robot_Walking_X-Walking_Robot_Movement.Act_Slice[4])<0.15 THEN
			// 到达目标位置,并且是六条腿支撑(state=2,realstate=3)的情况下,停止运动,并将User_Moving_Control复位
			IF Walking_Robot_Movement.state = 2 AND Walking_Robot_Movement.realState = 3 THEN
				// 先关使能信号,后关Enable和Disable两个外部运动开始信号
				User_Moving_Control := FALSE;
				Walking_Robot_Movement.ExtSetPointEnable 	:= FALSE;
				Walking_Robot_Movement.ExtSetPointDisable	:= TRUE;
			END_IF
		//ELSE
			//Walking_Robot_Movement.ExtSetPointEnable 		:= TRUE;
		END_IF
		
	END_IF
	
	
	// 不激活界面,因此界面所有的按钮默认关闭
ELSIF NOT Walking_Welding_Robot_Joint_Control THEN
	Walking_Welding_Robot_Power 			:= FALSE;
	Walking_Welding_Robot_Home_Execute 		:= FALSE;
	Walking_Welding_Robot_Moving_Execute	:= FALSE;
	User_Moving_Control						:= FALSE;
	Auto_Moving_Control						:= FALSE;
END_IF
END_ACTION

ACTION Variable_Monitor:
// =====================关键数据信号监测======================
END_ACTION

ACTION Variable_Set:

END_ACTION

END_PROGRAM

// ---- POUs/Welding_Arm_Control.TcPOU
PROGRAM Welding_Arm_Control

VAR CONSTANT
	MotorNum					: INT := 6;								// 接入控制的电机数量
END_VAR

VAR_INPUT
	// ====== 模块动作信号(按动作先后排列) ======
	Power_Execute 				: BOOL;									// 上电使能
	Axis_Power					: ARRAY[1..MotorNum] OF BOOL;			// 单电机上电
	Welding_Arm_Power			: BOOL;									// 焊接臂所有电机上电
	
	Home_Execute				: BOOL;									// 找零使能
	Axis_Home_Set				: ARRAY[1..MotorNum] OF BOOL;			// 单电机找零
	Welding_Arm_Home_Set		: BOOL;									// 焊接臂所有电机找零

	Reset_Execute				: BOOL;									// 电机驱动重置使能
	Axis_Reset					: ARRAY[1..MotorNum] OF BOOL;			// 单电机驱动重置
	Welding_Arm_Reset			: BOOL;									// 焊接臂整体电机驱动重置
	
	Welding_Arm_Move_Execute	: BOOL;									// 焊接臂运动程序使能	
	Move_Absolute_Execute		: BOOL;									// 绝对运动使能
	Move_Relative_Execute		: BOOL;									// 相对运动使能
	Axis_Absolute_Eable			: ARRAY[1..MotorNum] OF BOOL;			// 单电机绝对运动使能
	Axis_Relative_Eable			: ARRAY[1..MotorNum] OF BOOL;			// 单电机相对运动使能
	Axis_Move_Absolute_Position	: ARRAY[1..MotorNum] OF LREAL;			// 单电机绝对运动位置
	Axis_Move_Relative_Position	: ARRAY[1..MotorNum] OF LREAL;			// 单电机相对运动位置			
	
END_VAR
VAR
	// ====== NC轴变量 ======
	Axis_Welding_Arm			: ARRAY[1..MotorNum] OF Axis;			// 定义焊接臂轴参量(可以调整数据上限来调整电机数目)
	Axis_Number 				: INT;									// 定义轴数目
	
	// ====== 状态监测变量 ======
	Power_Status				: ARRAY[1..MotorNum] OF BOOL;			// 单电机上电状态
	Home_Done					: ARRAY[1..MotorNum] OF BOOL;			// 单电机找零状态
	Welding_Arm_Home_Done		: BOOL;									// 机器臂找零完成状态
	MoveAbsoluteDone			: ARRAY[1..MotorNum] OF BOOL;			// 单电机绝对运动状态
	MoveRelativeDone			: ARRAY[1..MotorNum] OF BOOL;			// 单电机相对运动状态
	
	Welding_Arm_Error			: BOOL;									// 焊接臂电机错误信号
	Axis_Error					: ARRAY[1..MotorNum] OF BOOL;			// 单电机错误信号
	Axis_ErrorID				: ARRAY[1..MotorNum] OF UDINT;			// 单电机错误码
	
	Axis_ActPostion				: ARRAY[1..MotorNum] OF LREAL;			// 单电机实际位置
	Axis_ActVelocity			: ARRAY[1..MotorNum] OF LREAL;			// 单电机实际速度
	
	Current_Turque_Value  AT%IW0: ARRAY[1..MotorNum] OF INT ;			// 单电机实际电流
	Digital_Inputs  	  AT%I* : ARRAY[1..MotorNum] OF DINT ;			// 驱动数字输入信号（Link到驱动器中的Digital Inputs）
	
	Home_Switch_value 			: ARRAY[1..MotorNum] OF BOOL;			// 限位开关值
	
	Max_Turque_Value 			: INT ;									// 最大电流边界值(机械限位法找零时用来判断运动极限位置)
END_VAR


Variable_Monitor();					// 变量监测程序

Logic_Control();					// 逻辑控制程序

Variable_Set();						// 变量设置程序

Welding_Arm_Action();				// 焊接臂整体运动程序

Welding_Arm_Single_Motor_Action();	// 焊接臂单电机运动程序

//Safety();							// 强安全措施程序

ACTION Logic_Control:
// =======================控制逻辑区==========================
// 保证所有的动作拥有合理的先后顺序，优化控制逻辑
// 也防止出现两个或两个以上动作同时进行的情况，保证控制安全

// ====== 电机驱动重置逻辑 ======
FOR Axis_Number := 1 TO MotorNum {BY 1} DO
	IF Axis_Error[Axis_Number] THEN
		Welding_Arm_Error := TRUE;
		EXIT;
	END_IF
	Welding_Arm_Error := FALSE;
END_FOR

IF Welding_Arm_Error THEN
	Reset_Execute := TRUE;
ELSIF NOT Welding_Arm_Error THEN
	Reset_Execute := FALSE;
END_IF

IF NOT Reset_Execute THEN
	FOR Axis_Number := 1 TO MotorNum {BY 1} DO
		Axis_Reset[Axis_Number] := FALSE;
		Axis_Welding_Arm[Axis_Number].Reset(Drive_Reset:= Axis_Reset[Axis_Number]);
	END_FOR
END_IF
	// 没有错误则不允许按按钮,或清除了错误按钮回弹
FOR Axis_Number := 1 TO MotorNum {BY 1} DO
	IF NOT Axis_Error[Axis_Number] THEN
		Axis_Reset[Axis_Number] := FALSE;
	END_IF
END_FOR

// ====== 上电逻辑 ======
IF NOT Power_Execute THEN
	FOR Axis_Number := 1 TO MotorNum {BY 1} DO
		Axis_Power[Axis_Number] := FALSE;
		Axis_Welding_Arm[Axis_Number].Power(Axis_Enable:= Axis_Power[Axis_Number]);
	END_FOR
END_IF

// ====== 找零逻辑 ======
IF Home_Execute THEN
	FOR Axis_Number := 1 TO MotorNum {BY 1} DO
		IF Home_Done[Axis_Number] THEN			// 	丝杠到达零点位置后，单电机标零使能位关闭			
			Axis_Home_Set[Axis_Number] := FALSE;	
			Axis_Welding_Arm[Axis_Number].Home_Sensor_Backward(	Drive_Home:= Axis_Home_Set[Axis_Number], 
													Home_Switch := NOT Home_Switch_value[Axis_Number]);
		END_IF
	END_FOR
	Move_Absolute_Execute := FALSE;							// 设定零点时，不能进行其他运动
	//ExSetPoint_Execute :=0;
ELSIF NOT Home_Execute THEN
	FOR Axis_Number := 1 TO MotorNum {BY 1} DO
		//Axis_Start_Back[Axis_Number] :=0;
		Axis_Home_Set[Axis_Number] := FALSE;
	END_FOR
END_IF

// ====== 绝对运动逻辑 ======
IF Move_Absolute_Execute THEN
	//Absolute_Eable := TRUE;
	Home_Execute := FALSE;							// 运动运动使能时，焊接臂调零必须结束
	//ExSetPoint_Execute :=0;						// 运动运动时，不能进行其他运动
	FOR Axis_Number := 1 TO MotorNum {BY 1} DO
		IF MoveAbsoluteDone[Axis_Number] THEN		// 	丝杠到达设定位置后，单电机绝对运动使能位关闭
			Axis_Absolute_Eable[Axis_Number] := FALSE;
		END_IF
	END_FOR
ELSIF NOT Move_Absolute_Execute THEN							// 运动不使能,轴不能运动
	FOR Axis_Number := 1 TO MotorNum {BY 1} DO
		Axis_Absolute_Eable[Axis_Number] := FALSE;
		Axis_Welding_Arm[Axis_Number].Move_Absolute(  Drive_Move_Absolute:= Axis_Absolute_Eable[Axis_Number], 
													  Absolute_Position:= Axis_Move_Absolute_Position[Axis_Number]);
	END_FOR
END_IF

// ====== 焊接臂相对运动逻辑 ======
IF Move_Relative_Execute THEN
	//Relative_Eable := TRUE;
	Home_Execute := FALSE;							// 运动运动使能时，焊接臂调零必须结束
	//ExSetPoint_Execute :=0;						// 运动运动时，不能进行其他运动
	FOR Axis_Number := 1 TO MotorNum {BY 1} DO
		IF MoveRelativeDone[Axis_Number] THEN		// 	丝杠到达设定位置后，单电机相对运动使能位关闭
			Axis_Relative_Eable[Axis_Number] := FALSE;
			Axis_Welding_Arm[Axis_Number].Move_Relative(  Drive_Move_Relative:= Axis_Relative_Eable[Axis_Number], 
													  Relative_Position:= Axis_Move_Relative_Position[Axis_Number]);
		END_IF
	END_FOR
ELSIF NOT Move_Relative_Execute THEN							// 运动不使能,轴不能运动
	FOR Axis_Number := 1 TO MotorNum {BY 1} DO
		Axis_Relative_Eable[Axis_Number] := FALSE;
		Axis_Welding_Arm[Axis_Number].Move_Relative(  Drive_Move_Relative:= Axis_Relative_Eable[Axis_Number], 
													  Relative_Position:= Axis_Move_Relative_Position[Axis_Number]);
	END_FOR
END_IF
END_ACTION

ACTION Safety:
// 保证丝杠行程和电机速度在规定范围内

// 如果没在找零，检测到焊接臂升降或径向关节接近开关信号即停止焊接臂上所有电机
IF NOT Home_Execute THEN
	// Digital_Inputs[1].19 为焊接臂升降电机接近开关(下)标识位
	// Digital_Inputs[3].20 为焊接臂径向电机接近开关(远离电机侧)标识位
	IF Digital_Inputs[1].18 OR Digital_Inputs[1].19 OR Digital_Inputs[3].20 OR Digital_Inputs[3].21 THEN
		FOR Axis_Number := 1 TO MotorNum {BY 1} DO
			//Axis_Power[Axis_Number] := FALSE;
		END_FOR
	END_IF
END_IF

//IF Digital_Inputs[1].18 THEN
//	pos_up := Axis_Welding_Arm[1].ActPosition;
//	range_v := pos_down - pos_up;
//	Axis_Power[1] := FALSE;
//END_IF
//IF Digital_Inputs[1].19 THEN
//	pos_down := Axis_Welding_Arm[1].ActPosition;
//	Axis_Move_Relative_Position[1] := -300;
//ELSE
//	Axis_Move_Relative_Position[1] := 200;
//END_IF

//IF Digital_Inputs[2].20 THEN
//	pos_far := Axis_Welding_Arm[2].ActPosition;
//	range_h := pos_far - pos_near;
//	Axis_Power[2] := FALSE;
//END_IF
//IF Digital_Inputs[2].21 THEN
//	pos_near := Axis_Welding_Arm[2].ActPosition;

//	Axis_Move_Relative_Position[2] := 200;
//ELSE
//	Axis_Move_Relative_Position[2] := 3;
//END_IF
END_ACTION

ACTION Variable_Monitor:
// =====================关键数据信号监测======================

// ====== 设置最大力矩(边界控制条件) ======
FOR Axis_Number := 1 TO MotorNum {BY 1} DO
	Axis_Welding_Arm[Axis_Number].Max_Turque_Value := Max_Turque_Value;
END_FOR

// ====== 检测实际力矩 ======
FOR Axis_Number := 1 TO MotorNum {BY 1} DO
	Axis_Welding_Arm[Axis_Number].Current_Turque_Value := Current_Turque_Value[Axis_Number];
END_FOR

// ====== 检测轴实际位置、速度 ======
FOR Axis_Number := 1 TO MotorNum {BY 1} DO
	Axis_ActPostion[Axis_Number] 	:= Axis_Welding_Arm[Axis_Number].ActPosition;
	Axis_ActVelocity[Axis_Number] 	:= Axis_Welding_Arm[Axis_Number].ActVelocity;
END_FOR

// ====== 检测上电状态 ======
FOR Axis_Number := 1 TO MotorNum {BY 1} DO
	Power_Status[Axis_Number] := Axis_Welding_Arm[Axis_Number].State_PowerStatus;
END_FOR

// ====== 检测找零状态 ======
FOR Axis_Number := 1 TO MotorNum {BY 1} DO
	Home_Done[Axis_Number] := Axis_Welding_Arm[Axis_Number].State_HomeDone;
END_FOR

// ====== 检测电机绝对运动状态 ======
FOR Axis_Number := 1 TO MotorNum {BY 1} DO
	MoveAbsoluteDone[Axis_Number] := Axis_Welding_Arm[Axis_Number].State_MoveAbsoluteDone;
END_FOR

// ====== 检测电机相对运动状态 ======
FOR Axis_Number := 1 TO MotorNum {BY 1} DO
	MoveRelativeDone[Axis_Number] := Axis_Welding_Arm[Axis_Number].State_MoveRelativeDone;
END_FOR

// ====== 检测电机错误 ======
FOR Axis_Number := 1 TO MotorNum {BY 1} DO
	Axis_Error[Axis_Number] 	:= Axis_Welding_Arm[Axis_Number].Axis_Error;
	Axis_ErrorID[Axis_Number] 	:= Axis_Welding_Arm[Axis_Number].Axis_ErrorID;
END_FOR
END_ACTION

ACTION Variable_Set:
// ====== 设置速度 ======
FOR Axis_Number := 1 TO MotorNum {BY 1} DO							//此时每一个电机的速度都是一样的
	Axis_Welding_Arm[Axis_Number].Home_Velocity 	:= 5;			//找零速度(Axis_Jog中的速度)
	Axis_Welding_Arm[Axis_Number].Move_Relative_Velocity	:=5;	//相对运动速度
END_FOR
IF Home_Execute THEN
	FOR Axis_Number := 1 TO MotorNum {BY 1} DO
		Axis_Welding_Arm[Axis_Number].Move_Absolute_Velocity := 5;	//找零之后运动至轨迹起始点的速度
	END_FOR
ELSE
	FOR Axis_Number := 1 TO MotorNum {BY 1} DO
			Axis_Welding_Arm[Axis_Number].Move_Absolute_Velocity	:=10;
	END_FOR
END_IF
	

// ====== 设置绝对运动位置 ======
FOR Axis_Number := 1 TO MotorNum {BY 1} DO
	Axis_Move_Absolute_Position[Axis_Number] := 100;
END_FOR

// ====== 设置相对运动距离 ======
FOR Axis_Number := 1 TO MotorNum {BY 1} DO
	Axis_Move_Relative_Position[Axis_Number] := -15;
END_FOR

// ====== 设置最大力矩(找零过程判断已到丝杠顶点) ======
Max_Turque_Value := 1400;

// ====== 设置电机设零后到达Simulink模型初始位置 ======
IF Home_Execute THEN
	FOR Axis_Number := 1 TO MotorNum {BY 1} DO
		Axis_Welding_Arm[Axis_Number].Home_Absolute_Position := Welding_Arm_Movement.ExSetPoint_Position[Axis_Number];
	END_FOR
END_IF
END_ACTION

ACTION Welding_Arm_Action:
// =================焊接臂整体运动命令区======================
// 六足所有电机整体控制

// ====== 焊接臂所有电机驱动重置 ======
IF Welding_Arm_Reset THEN							// 缺少输入
	IF Reset_Execute THEN
		FOR Axis_Number := 1 TO MotorNum {BY 1} DO
			Axis_Reset[Axis_Number] := TRUE;
			Axis_Welding_Arm[Axis_Number].Reset(Drive_Reset:= Axis_Reset[Axis_Number]);
		END_FOR
	END_IF
END_IF	

// ====== 焊接臂所有电机上电 ======
IF Welding_Arm_Power THEN	
	IF Power_Execute THEN
		FOR Axis_Number := 1 TO MotorNum {BY 1} DO
			Axis_Power[Axis_Number] := TRUE ;
		END_FOR
	END_IF
END_IF
	
// ====== 焊接臂所有电机找零 ======
IF Welding_Arm_Home_Set THEN
	IF Home_Execute THEN
		FOR Axis_Number := 1 TO MotorNum {BY 1} DO
			IF NOT Home_Done[Axis_Number] THEN
				Axis_Home_Set[Axis_Number] := TRUE;
				Axis_Welding_Arm[Axis_Number].Home_Sensor_Backward(	Drive_Home:= Axis_Home_Set[Axis_Number], 
													Home_Switch := NOT Home_Switch_value[Axis_Number]);
			ELSIF Home_Done[Axis_Number] THEN
				Axis_Home_Set[Axis_Number] := FALSE;
				Axis_Welding_Arm[Axis_Number].Home_Sensor_Backward(	Drive_Home:= Axis_Home_Set[Axis_Number], 
													Home_Switch := NOT Home_Switch_value[Axis_Number]);
			END_IF
		END_FOR
	ELSIF NOT Home_Execute THEN
		FOR Axis_Number := 1 TO MotorNum {BY 1} DO
			Axis_Home_Set[Axis_Number] := FALSE;
		END_FOR
	END_IF
ELSIF NOT Welding_Arm_Home_Set AND NOT Home_Execute THEN
	FOR Axis_Number := 1 TO MotorNum {BY 1} DO
		Axis_Home_Set[Axis_Number] := FALSE;
	END_FOR
END_IF

IF Home_Execute THEN
	IF ABS(Welding_Arm_Movement.ExSetPoint_Position[1]-Axis_ActPostion[1]) < 0.1 AND
		ABS(Welding_Arm_Movement.ExSetPoint_Position[2]-Axis_ActPostion[2]) < 0.1 AND
		 ABS(Welding_Arm_Movement.ExSetPoint_Position[3]-Axis_ActPostion[3]) < 0.1 AND
		  ABS(Welding_Arm_Movement.ExSetPoint_Position[4]-Axis_ActPostion[4]) < 0.1 AND
		   ABS(Welding_Arm_Movement.ExSetPoint_Position[5]-Axis_ActPostion[5]) < 0.1 AND
			ABS(Welding_Arm_Movement.ExSetPoint_Position[6]-Axis_ActPostion[6]) < 0.1 THEN
		Welding_Arm_Home_Done := TRUE;
	END_IF
ELSIF NOT Home_Execute THEN
	Welding_Arm_Home_Done := FALSE;
END_IF

// ====== 焊接臂所有电机绝对运动 ======
IF Welding_Arm_Move_Execute THEN
	IF Move_Absolute_Execute THEN
		FOR Axis_Number := 1 TO MotorNum {BY 1} DO
			IF MoveAbsoluteDone[Axis_Number] THEN		// 	丝杠到达设定位置后，单电机绝对运动使能位关闭
				Axis_Absolute_Eable[Axis_Number] := FALSE;
			ELSE
				Axis_Absolute_Eable[Axis_Number] := TRUE;
			END_IF
		END_FOR
	END_IF
ELSIF NOT Welding_Arm_Move_Execute AND NOT Move_Absolute_Execute THEN 
	FOR Axis_Number := 1 TO MotorNum {BY 1} DO
		Axis_Absolute_Eable[Axis_Number] := FALSE;
	END_FOR
END_IF

// ====== 焊接臂所有电机相对运动 ======
IF Welding_Arm_Move_Execute THEN
	IF Move_Relative_Execute THEN
		FOR Axis_Number := 1 TO MotorNum {BY 1} DO
			IF MoveRelativeDone[Axis_Number] THEN		// 	丝杠到达设定位置后，单电机相对运动使能位关闭
				Axis_Relative_Eable[Axis_Number] := FALSE;
			ELSE
				Axis_Relative_Eable[Axis_Number] := TRUE;
			END_IF
		END_FOR
	END_IF
ELSIF NOT Welding_Arm_Move_Execute AND NOT Move_Relative_Execute THEN 
	FOR Axis_Number := 1 TO MotorNum {BY 1} DO
		Axis_Relative_Eable[Axis_Number] := FALSE;
	END_FOR
END_IF
END_ACTION

ACTION Welding_Arm_Single_Motor_Action:

// ====== 单电机驱动重置 ======
IF Reset_Execute THEN
	FOR Axis_Number := 1 TO MotorNum {BY 1} DO
		Axis_Welding_Arm[Axis_Number].Reset(Drive_Reset:= Axis_Reset[Axis_Number]);
	END_FOR
END_IF

// ====== 单电机上电 ======
IF Power_Execute THEN
	FOR Axis_Number := 1 TO MotorNum {BY 1} DO
		Axis_Welding_Arm[Axis_Number].Power(Axis_Enable:= Axis_Power[Axis_Number]);
	END_FOR
END_IF

// ====== 单电机找零 ======
IF Home_Execute THEN
	// 如果用模型控制，必须加上下面一句话
	FOR Axis_Number := 1 TO MotorNum {BY 1} DO
		IF Axis_Number = 3 THEN
			Home_Switch_value[Axis_Number] := Digital_Inputs[Axis_Number].21;		// 焊接臂径向电机接近开关(靠近电机侧)标识位
		ELSE
			Home_Switch_value[Axis_Number] := Digital_Inputs[Axis_Number].18;
		END_IF
		
		Axis_Welding_Arm[Axis_Number].Home_Sensor_Backward(	Drive_Home:= Axis_Home_Set[Axis_Number], 
													Home_Switch := Home_Switch_value[Axis_Number]);
	END_FOR
END_IF

// ====== 单电机绝对移动 ======
IF Move_Absolute_Execute THEN
	FOR Axis_Number := 1 TO MotorNum {BY 1} DO
		Axis_Welding_Arm[Axis_Number].Move_Absolute(	Drive_Move_Absolute:= Axis_Absolute_Eable[Axis_Number], 
														Absolute_Position:= Axis_Move_Absolute_Position[Axis_Number]);
	END_FOR
END_IF

// ====== 单电机相对移动 ======
IF Move_Relative_Execute THEN
	FOR Axis_Number := 1 TO MotorNum {BY 1} DO
		Axis_Welding_Arm[Axis_Number].Move_Relative(	Drive_Move_Relative:= Axis_Relative_Eable[Axis_Number], 
														Relative_Position:= Axis_Move_Relative_Position[Axis_Number]);
	END_FOR
END_IF
END_ACTION

END_PROGRAM

// ---- POUs/Welding_Arm_Movement.TcPOU
PROGRAM Welding_Arm_Movement

VAR CONSTANT
	MotorNum			: INT := 6;
END_VAR

VAR_INPUT
	ExSetPoint_Execute	: BOOL;					// 机器人外部信号发生使能
	ExtSetPointEnable	: BOOL;					// 外部信号发生信号
	ExtSetPointDisable	: BOOL;					// 外部信号结束信号
END_VAR

VAR
	Axis_Number			: INT;					// 轴数量,用来遍历轴	
	
	// ====== 定义Simulink模块 ======
	Welding_Arm_Simulink: FB_WeldingArm6AxisMotion_Control(oid:=16#01010050);	// Simulink模型定义
	
		// Simulink输入
	t_Interval			: LREAL := 0.001;		// 取样时间间隔，默认为1ms
	t					: LREAL := 0;			// 取样当前时间变量，以0为起点
		// Simulink输出
	T_ALL				: LREAL := 100;			// Simulink模型运动总时长
	ExSetPoint_Position	: ARRAY[1..6] OF LREAL;// 外部信号位置
END_VAR


Variable_Monitor();			// 变量监测程序

Logic_Control();			// 逻辑控制程序

Variable_Set();				// 变量设置程序

ExSetPoint_Action();		// 外部发生运动程序

//Safety();					// 强安全措施

ACTION ExSetPoint_Action:

// ====== Simulink激活与外部信号运动 ======
IF ExSetPoint_Execute OR Welding_Arm_Control.Home_Execute THEN
	// Simulink激活
	Welding_Arm_Simulink.Execute();	
	// 外部信号运动开始
	FOR Axis_Number := 1 TO Welding_Arm_Control.MotorNum {BY 1} DO
		Welding_Arm_Control.Axis_Welding_Arm[Axis_Number].ExtSetPoint(Drive_ExtSetPointEnable:= ExtSetPointEnable, 
											Drive_ExtSetPointDisable:= ExtSetPointDisable, 
											ExSetPosition:= ExSetPoint_Position[Axis_Number]);
	END_FOR
END_IF

// ====== 采样时间 =======
IF ExtSetPointEnable THEN
	t := t + t_Interval;
	ExtSetPointDisable 	:= FALSE;
END_IF

IF t>=T_ALL THEN
	ExtSetPointEnable 	:= FALSE;
	t := 0;
	ExtSetPointDisable 	:= TRUE;
END_IF
END_ACTION

ACTION Logic_Control:
// =======================控制逻辑区==========================
// 保证所有的动作拥有合理的先后顺序，优化控制逻辑
// 也防止出现两个或两个以上动作同时进行的情况，保证控制安全

// =====================外部信号发生逻辑========================
IF ExSetPoint_Execute THEN
	Welding_Arm_Control.Home_Execute := FALSE;						// 外部信号发生使能时，机器人调零必须结束
ELSIF NOT ExSetPoint_Execute THEN
	ExtSetPointEnable := 0;						// 外部信号发生不使能时，外部信号不能进入程序
	ExtSetPointDisable :=0;
ELSIF ExtSetPointDisable THEN
	ExtSetPointEnable :=0;						// 外部信号发生停止与外部信号发生开始不能同时进行
END_IF


IF Welding_Arm_Control.Home_Execute OR Welding_Arm_Control.Move_Absolute_Execute OR Welding_Arm_Control.Move_Relative_Execute THEN
	ExSetPoint_Execute := FALSE;
END_IF
END_ACTION

ACTION Safety:
// 保证丝杠行程和电机速度在规定范围内

// 如果没在找零，检测到焊接臂升降或径向关节接近开关信号即停止焊接臂上所有电机

//IF Digital_Inputs[1].18 THEN
//	pos_up := Axis_Welding_Arm[1].ActPosition;
//	range_v := pos_down - pos_up;
//	Axis_Power[1] := FALSE;
//END_IF
//IF Digital_Inputs[1].19 THEN
//	pos_down := Axis_Welding_Arm[1].ActPosition;
//	Axis_Move_Relative_Position[1] := -300;
//ELSE
//	Axis_Move_Relative_Position[1] := 200;
//END_IF

//IF Digital_Inputs[2].20 THEN
//	pos_far := Axis_Welding_Arm[2].ActPosition;
//	range_h := pos_far - pos_near;
//	Axis_Power[2] := FALSE;
//END_IF
//IF Digital_Inputs[2].21 THEN
//	pos_near := Axis_Welding_Arm[2].ActPosition;

//	Axis_Move_Relative_Position[2] := 200;
//ELSE
//	Axis_Move_Relative_Position[2] := 3;
//END_IF
END_ACTION

ACTION Variable_Monitor:
// =====================关键数据信号监测======================
END_ACTION

ACTION Variable_Set:
// ===================程序与模型的变量链接===================

	// -- 输入 -- 
Welding_Arm_Simulink.stInput.t := t;								// 采样时间t与Simulink模型中的采样时间链接

	// -- 输出 -- 
T_ALL := Welding_Arm_Simulink.stOutput.T_ALL;
FOR Axis_Number := 1 TO MotorNum {BY 1} DO
	ExSetPoint_Position[Axis_Number] := Welding_Arm_Simulink.stOutput.Disp_J[Axis_Number-1]; // Simulink中的电机输出位移输入到控制模型
END_FOR
END_ACTION

END_PROGRAM

// ---- DUTs/Welding_Arm_Simulink/FB_WeldingArm6AxisMotion_Control.TcPOU
{attribute 'TcDependOnClassFactory' := 'WeldingArm6AxisMotion_Control'}
FUNCTION_BLOCK FB_WeldingArm6AxisMotion_Control EXTENDS FB_TcMatSimObject
VAR_INPUT
	stInput: ST_WeldingArm6AxisMotion_Control_Input;
END_VAR
VAR_OUTPUT
	stOutput: ST_WeldingArm6AxisMotion_Control_Output;
END_VAR
VAR
	stInitData: ST_WeldingArm6AxisMotion_Control_InitData;
	arrDataAreas: ARRAY[1..2] OF ST_TcMatSimObjectDataAreaInfo;
	bParametersVerified: BOOL;
END_VAR

PROPERTY CallBy_Online : TctModuleCallByType
GET
hResult := GetObjPara(16#00000000,sizeof(CallBy_Online),adr(CallBy_Online));
END_GET
SET
hResult := SetObjPara(16#00000000,sizeof(CallBy_Online),adr(CallBy_Online));
END_SET
END_PROPERTY

PROPERTY CallBy_Startup : TctModuleCallByType
GET
CallBy_Startup := stInitData.CallBy;
END_GET
SET
stInitData.CallBy := CallBy_Startup;
END_SET
END_PROPERTY

PROPERTY ContextInfoArr_0_TaskCycleTimeNs_Online : UDINT
GET
hResult := GetObjPara(16#03002080,sizeof(ContextInfoArr_0_TaskCycleTimeNs_Online),adr(ContextInfoArr_0_TaskCycleTimeNs_Online));
END_GET
SET
hResult := SetObjPara(16#03002080,sizeof(ContextInfoArr_0_TaskCycleTimeNs_Online),adr(ContextInfoArr_0_TaskCycleTimeNs_Online));
END_SET
END_PROPERTY

PROPERTY ContextInfoArr_0_TaskCycleTimeNs_Startup : UDINT
GET
ContextInfoArr_0_TaskCycleTimeNs_Startup := stInitData.ContextInfoArr_0_TaskCycleTimeNs;
END_GET
SET
stInitData.ContextInfoArr_0_TaskCycleTimeNs := ContextInfoArr_0_TaskCycleTimeNs_Startup;
END_SET
END_PROPERTY

PROPERTY ContextInfoArr_0_TaskOid_Online : OTCID
GET
hResult := GetObjPara(16#03002060,sizeof(ContextInfoArr_0_TaskOid_Online),adr(ContextInfoArr_0_TaskOid_Online));
END_GET
SET
hResult := SetObjPara(16#03002060,sizeof(ContextInfoArr_0_TaskOid_Online),adr(ContextInfoArr_0_TaskOid_Online));
END_SET
END_PROPERTY

PROPERTY ContextInfoArr_0_TaskOid_Startup : OTCID
GET
ContextInfoArr_0_TaskOid_Startup := stInitData.ContextInfoArr_0_TaskOid;
END_GET
SET
stInitData.ContextInfoArr_0_TaskOid := ContextInfoArr_0_TaskOid_Startup;
END_SET
END_PROPERTY

PROPERTY ContextInfoArr_0_TaskPort_Online : UINT
GET
hResult := GetObjPara(16#03002090,sizeof(ContextInfoArr_0_TaskPort_Online),adr(ContextInfoArr_0_TaskPort_Online));
END_GET
SET
hResult := SetObjPara(16#03002090,sizeof(ContextInfoArr_0_TaskPort_Online),adr(ContextInfoArr_0_TaskPort_Online));
END_SET
END_PROPERTY

PROPERTY ContextInfoArr_0_TaskPort_Startup : UINT
GET
ContextInfoArr_0_TaskPort_Startup := stInitData.ContextInfoArr_0_TaskPort;
END_GET
SET
stInitData.ContextInfoArr_0_TaskPort := ContextInfoArr_0_TaskPort_Startup;
END_SET
END_PROPERTY

PROPERTY ContextInfoArr_0_TaskPriority_Online : UDINT
GET
hResult := GetObjPara(16#03002070,sizeof(ContextInfoArr_0_TaskPriority_Online),adr(ContextInfoArr_0_TaskPriority_Online));
END_GET
SET
hResult := SetObjPara(16#03002070,sizeof(ContextInfoArr_0_TaskPriority_Online),adr(ContextInfoArr_0_TaskPriority_Online));
END_SET
END_PROPERTY

PROPERTY ContextInfoArr_0_TaskPriority_Startup : UDINT
GET
ContextInfoArr_0_TaskPriority_Startup := stInitData.ContextInfoArr_0_TaskPriority;
END_GET
SET
stInitData.ContextInfoArr_0_TaskPriority := ContextInfoArr_0_TaskPriority_Startup;
END_SET
END_PROPERTY

PROPERTY ContextInfoArr_0_TaskSortOrder_Online : UDINT
GET
hResult := GetObjPara(16#030020b0,sizeof(ContextInfoArr_0_TaskSortOrder_Online),adr(ContextInfoArr_0_TaskSortOrder_Online));
END_GET
SET
hResult := SetObjPara(16#030020b0,sizeof(ContextInfoArr_0_TaskSortOrder_Online),adr(ContextInfoArr_0_TaskSortOrder_Online));
END_SET
END_PROPERTY

PROPERTY ContextInfoArr_0_TaskSortOrder_Startup : UDINT
GET
ContextInfoArr_0_TaskSortOrder_Startup := stInitData.ContextInfoArr_0_TaskSortOrder;
END_GET
SET
stInitData.ContextInfoArr_0_TaskSortOrder := ContextInfoArr_0_TaskSortOrder_Startup;
END_SET
END_PROPERTY

PROPERTY CycleUpdateExecuted_Online : BOOL
GET
hResult := GetObjPara(16#00000004,sizeof(CycleUpdateExecuted_Online),adr(CycleUpdateExecuted_Online));
END_GET
SET
hResult := SetObjPara(16#00000004,sizeof(CycleUpdateExecuted_Online),adr(CycleUpdateExecuted_Online));
END_SET
END_PROPERTY

METHOD Execute : HRESULT

IF (SUCCEEDED(hResult)) THEN
  hResult := VerifyParameters();
END_IF

	// update DataArea information
SetDataAreaInfo(ADR(arrDataAreas),2);
	
	// call base method
Execute := SUPER^.Execute();
END_METHOD

PROPERTY ExecuteModelCode_Online : BOOL
GET
hResult := GetObjPara(16#00000008,sizeof(ExecuteModelCode_Online),adr(ExecuteModelCode_Online));
END_GET
SET
hResult := SetObjPara(16#00000008,sizeof(ExecuteModelCode_Online),adr(ExecuteModelCode_Online));
END_SET
END_PROPERTY

PROPERTY ExecuteModelCode_Startup : BOOL
GET
ExecuteModelCode_Startup := stInitData.ExecuteModelCode;
END_GET
SET
stInitData.ExecuteModelCode := ExecuteModelCode_Startup;
END_SET
END_PROPERTY

PROPERTY ExecutionSequence_Online : TctModuleExecutionSequenceType
GET
hResult := GetObjPara(16#00000001,sizeof(ExecutionSequence_Online),adr(ExecutionSequence_Online));
END_GET
SET
hResult := SetObjPara(16#00000001,sizeof(ExecutionSequence_Online),adr(ExecutionSequence_Online));
END_SET
END_PROPERTY

PROPERTY ExecutionSequence_Startup : TctModuleExecutionSequenceType
GET
ExecutionSequence_Startup := stInitData.ExecutionSequence;
END_GET
SET
stInitData.ExecutionSequence := ExecutionSequence_Startup;
END_SET
END_PROPERTY

METHOD FB_init : BOOL
VAR_INPUT
	/// if TRUE, the retain variables are initialized (warm start / cold start)
	bInitRetains: BOOL;
	/// if TRUE, the instance afterwards gets moved into the copy code (online change)
	bInCopyCode: BOOL;
	oid: OTCID;
END_VAR
VAR
	clsId: CLSID;
END_VAR

// initialize flags
bParametersVerified := false;
                    
// set module class id for compatibility check
clsId.Data1 := 16#412caec1;
clsId.Data2 := 16#7008;
clsId.Data3 := 16#47ed;
clsId.Data4[0] := 16#9b;
clsId.Data4[1] := 16#82;
clsId.Data4[2] := 16#ce;
clsId.Data4[3] := 16#15;
clsId.Data4[4] := 16#e3;
clsId.Data4[5] := 16#d3;
clsId.Data4[6] := 16#23;
clsId.Data4[7] := 16#f9;

AssignClassId(clsId);
                    
// initialize InitData structure with default values              
stInitData.CallByHdr.indexGroup := 0;
stInitData.CallByHdr.indexOffset := 16#00000000;
stInitData.CallByHdr.cbData := SIZEOF(stInitData.CallBy);
stInitData.CallBy := TctModuleCallByType.Module;
stInitData.ExecutionSequenceHdr.indexGroup := 0;
stInitData.ExecutionSequenceHdr.indexOffset := 16#00000001;
stInitData.ExecutionSequenceHdr.cbData := SIZEOF(stInitData.ExecutionSequence);
stInitData.ExecutionSequence := TctModuleExecutionSequenceType.StateUpdateAfterOutputMapping;
stInitData.StepSizeHdr.indexGroup := 0;
stInitData.StepSizeHdr.indexOffset := 16#00000002;
stInitData.StepSizeHdr.cbData := SIZEOF(stInitData.StepSize);
stInitData.StepSize := TctStepSizeType.UseTaskCycleTime;
stInitData.ExecuteModelCodeHdr.indexGroup := 0;
stInitData.ExecuteModelCodeHdr.indexOffset := 16#00000008;
stInitData.ExecuteModelCodeHdr.cbData := SIZEOF(stInitData.ExecuteModelCode);
stInitData.ExecuteModelCode := 1;
stInitData.ModelParametersHdr.indexGroup := 0;
stInitData.ModelParametersHdr.indexOffset := 16#82000000;
stInitData.ModelParametersHdr.cbData := SIZEOF(stInitData.ModelParameters);
stInitData.ModelParameters.tcycle_Value := 5.00000000000000000e+00;
stInitData.ModelParameters.J1rg_Value[0] := 2.00000000000000000e+01;
stInitData.ModelParameters.J1rg_Value[1] := 2.00000000000000000e+02;
stInitData.ModelParameters.J2rg_Value[0] := -2.70000000000000000e+02;
stInitData.ModelParameters.J2rg_Value[1] := 9.00000000000000000e+01;
stInitData.ModelParameters.J3rg_Value[0] := 2.00000000000000000e+01;
stInitData.ModelParameters.J3rg_Value[1] := 1.30000000000000000e+02;
stInitData.ModelParameters.phirg_Value[0] := -3.00000000000000000e+01;
stInitData.ModelParameters.phirg_Value[1] := 3.00000000000000000e+01;
stInitData.ModelParameters.gamarg_Value[0] := 1.50000000000000000e+01;
stInitData.ModelParameters.gamarg_Value[1] := 3.50000000000000000e+01;
stInitData.ContextInfoArr_0_TaskOidHdr.indexGroup := 0;
stInitData.ContextInfoArr_0_TaskOidHdr.indexOffset := 16#03002060;
stInitData.ContextInfoArr_0_TaskOidHdr.cbData := SIZEOF(stInitData.ContextInfoArr_0_TaskOid);
stInitData.ContextInfoArr_0_TaskPriorityHdr.indexGroup := 0;
stInitData.ContextInfoArr_0_TaskPriorityHdr.indexOffset := 16#03002070;
stInitData.ContextInfoArr_0_TaskPriorityHdr.cbData := SIZEOF(stInitData.ContextInfoArr_0_TaskPriority);
stInitData.ContextInfoArr_0_TaskCycleTimeNsHdr.indexGroup := 0;
stInitData.ContextInfoArr_0_TaskCycleTimeNsHdr.indexOffset := 16#03002080;
stInitData.ContextInfoArr_0_TaskCycleTimeNsHdr.cbData := SIZEOF(stInitData.ContextInfoArr_0_TaskCycleTimeNs);
stInitData.ContextInfoArr_0_TaskPortHdr.indexGroup := 0;
stInitData.ContextInfoArr_0_TaskPortHdr.indexOffset := 16#03002090;
stInitData.ContextInfoArr_0_TaskPortHdr.cbData := SIZEOF(stInitData.ContextInfoArr_0_TaskPort);
stInitData.ContextInfoArr_0_TaskSortOrderHdr.indexGroup := 0;
stInitData.ContextInfoArr_0_TaskSortOrderHdr.indexOffset := 16#030020b0;
stInitData.ContextInfoArr_0_TaskSortOrderHdr.cbData := SIZEOF(stInitData.ContextInfoArr_0_TaskSortOrder);
stInitData.Header.cbData := SIZEOF(stInitData)-SIZEOF(stInitData.Header);
stInitData.Header.uiElmCnt := 10;


// set pointer to InitData structure
SetInitDataInfo(ADR(stInitData));

// set DataArea information
SetDataAreaInfo(ADR(arrDataAreas),2);
arrDataAreas[1].nDataAreaId := 0;
arrDataAreas[1].nSize := SIZEOF(stInput);
arrDataAreas[1].pPlcVar := ADR(stInput);
arrDataAreas[1].pModuleProcImg := 0;
arrDataAreas[1].eDataAreaType := E_TcMatSimDataAreaType.InputDst;
arrDataAreas[2].nDataAreaId := 1;
arrDataAreas[2].nSize := SIZEOF(stOutput);
arrDataAreas[2].pPlcVar := ADR(stOutput);
arrDataAreas[2].pModuleProcImg := 0;
arrDataAreas[2].eDataAreaType := E_TcMatSimDataAreaType.OutputSrc;


// initialize basic interface pointers and return
FB_init := SUCCEEDED(Init(oid));
END_METHOD

PROPERTY InitData : ST_WeldingArm6AxisMotion_Control_InitData
GET
InitData := stInitData;
END_GET
SET
stInitData := InitData;
END_SET
END_PROPERTY

PROPERTY Input_Online : ExtU_weldingArm6axisMotionTes_T
GET
hResult := GetObjPara(16#80000000,sizeof(Input_Online),adr(Input_Online));
END_GET
SET
hResult := SetObjPara(16#80000000,sizeof(Input_Online),adr(Input_Online));
END_SET
END_PROPERTY

{attribute 'object_name' := 'Internal_SetObjState'}
METHOD PROTECTED Internal_SetObjState
VAR_INPUT
	hr: REFERENCE TO HRESULT;
	nextState: TCOM_STATE;
END_VAR

// update pointer to InitData structure
SetInitDataInfo(ADR(stInitData));
// call base method
SUPER^.Internal_SetObjState(hr,nextState);
END_METHOD

PROPERTY MdlInitialized_Online : BOOL
GET
hResult := GetObjPara(16#00000003,sizeof(MdlInitialized_Online),adr(MdlInitialized_Online));
END_GET
SET
hResult := SetObjPara(16#00000003,sizeof(MdlInitialized_Online),adr(MdlInitialized_Online));
END_SET
END_PROPERTY

PROPERTY ModelParameters_Online : P_weldingArm6axisMotionTest1_T
GET
hResult := GetObjPara(16#82000000,sizeof(ModelParameters_Online),adr(ModelParameters_Online));
END_GET
SET
hResult := SetObjPara(16#82000000,sizeof(ModelParameters_Online),adr(ModelParameters_Online));
END_SET
END_PROPERTY

PROPERTY ModelParameters_Startup : P_weldingArm6axisMotionTest1_T
GET
ModelParameters_Startup := stInitData.ModelParameters;
END_GET
SET
stInitData.ModelParameters := ModelParameters_Startup;
END_SET
END_PROPERTY

PROPERTY ModuleBuildInfo_Online : TctModuleBuildInfoType
GET
hResult := GetObjPara(16#00000007,sizeof(ModuleBuildInfo_Online),adr(ModuleBuildInfo_Online));
END_GET
SET
hResult := SetObjPara(16#00000007,sizeof(ModuleBuildInfo_Online),adr(ModuleBuildInfo_Online));
END_SET
END_PROPERTY

PROPERTY ModuleInfo_Online : TctModuleInfoType
GET
hResult := GetObjPara(16#00000006,sizeof(ModuleInfo_Online),adr(ModuleInfo_Online));
END_GET
SET
hResult := SetObjPara(16#00000006,sizeof(ModuleInfo_Online),adr(ModuleInfo_Online));
END_SET
END_PROPERTY

{attribute 'object_name' := 'SaveOnlineParametersForInit'}
METHOD SaveOnlineParametersForInit : HRESULT
VAR
	idx: UINT;
	pInitElemHdr: POINTER TO TComInitDataElmHdr;
	pData: PVOID;
	nData: UDINT;
END_VAR
VAR CONSTANT
	nInitDataAlignment: UDINT := 4;
END_VAR

// update pointer to InitData structure
SetInitDataInfo(ADR(stInitData));
// call base method
SaveOnlineParametersForInit := SUPER^.SaveOnlineParametersForInit();
END_METHOD

PROPERTY SimulinkTime_Online : LREAL
GET
hResult := GetObjPara(16#00000005,sizeof(SimulinkTime_Online),adr(SimulinkTime_Online));
END_GET
SET
hResult := SetObjPara(16#00000005,sizeof(SimulinkTime_Online),adr(SimulinkTime_Online));
END_SET
END_PROPERTY

PROPERTY StepSize_Online : TctStepSizeType
GET
hResult := GetObjPara(16#00000002,sizeof(StepSize_Online),adr(StepSize_Online));
END_GET
SET
hResult := SetObjPara(16#00000002,sizeof(StepSize_Online),adr(StepSize_Online));
END_SET
END_PROPERTY

PROPERTY StepSize_Startup : TctStepSizeType
GET
StepSize_Startup := stInitData.StepSize;
END_GET
SET
stInitData.StepSize := StepSize_Startup;
END_SET
END_PROPERTY

{attribute 'object_name' := 'VerifyParameters'}
METHOD PRIVATE VerifyParameters : HRESULT
VAR
	moduleCallByParam: TctModuleCallByType;
END_VAR

IF (bParametersVerified) THEN
  VerifyParameters := Tc2_System.E_HRESULTAdsErr.HRESULT_ADS_NOERROR;
ELSE
  VerifyParameters := GetObjPara(stInitData.CallByHdr.indexOffset,SIZEOF(moduleCallByParam),ADR(moduleCallByParam));
  
  // check the "CallBy" parameter to be set to "Module"
  IF (SUCCEEDED(VerifyParameters) AND (moduleCallByParam <> TctModuleCallByType.Module)) THEN
      VerifyParameters := Tc2_System.E_HRESULTAdsErr.INVALIDPARM;
  END_IF
  
  // set the parameters verified flag
  bParametersVerified := SUCCEEDED(VerifyParameters);
END_IF
END_METHOD

END_FUNCTION_BLOCK

// ---- POUs/SignalData_Interface.TcPOU
PROGRAM SignalData_Interface
VAR_INPUT
	// ===================激光输入控制信号区==========
	enableScan			: BOOL;								// 开始激光扫描信号
	
	// ===================陀螺仪信号区==========
	open_windows 	AT 	%MD7 : BOOL;						// 控制传感器窗口的开关信号
END_VAR
VAR
	
	// ===================激光信号区==========
	Trigger: BOOL;												// The trigger for profile sensor
	
	LScanCounts			: INT;								// 已完成的激光线轮廓扫描数
	ScanTon				: TON;								// 扫描上升沿计时器
	ScanT				: TIME := T#2000MS;					// 扫描上升沿之后的高电平保持时间
	Digital_Outputs_16	: BOOL;
	
	pos_up				: LREAL;
	pos_down			: LREAL;
	range_v				: LREAL;
	pos_far				: LREAL;
	pos_near			: LREAL;
	range_h				: LREAL;
END_VAR
VAR_OUTPUT
	// ===================陀螺仪信号区==========
	W  		AT  %MD0 	: REAL;
	X		AT 	%MD1 	: REAL;
	Y		AT 	%MD2 	: REAL;
	Z		AT 	%MD3 	: REAL;
	ROLL 	AT 	%MD4 	: REAL;
	PITCH	AT 	%MD5 	: REAL;
	YAW		AT 	%MD6 	: REAL;
	
	// ===================激光信号控制区==========
	Welding_Arm_Digital_Outputs AT%Q* : DINT;					// 数字输出信号（Link到驱动器中的Digital Outputs）
END_VAR

VAR CONSTANT	
	LScanStepSize		: LREAL := 5;							// 激光扫描步长（LaserScanStepSize），对应电机转角（测试代码）
	LScanRange			: LREAL := 360;							// 激光扫描范围（LaserScanRange），对应电机总转角（测试代码）
END_VAR

Laser_Scan();
Signal_Monitor();

ACTION Laser_Scan:
// =================线激光测量触发信号生成程序===================
ScanTon(IN:= enableScan , PT:= ScanT , Q=> , ET=> );

IF Trigger AND (NOT Welding_Arm_Control.MoveRelativeDone[1]) AND (NOT Welding_Arm_Digital_Outputs.16)THEN
	Welding_Arm_Control.Axis_Relative_Eable[1] := TRUE;
END_IF


IF NOT Welding_Arm_Control.Axis_Relative_Eable[1] AND Trigger THEN
	enableScan := TRUE;
ELSE
	enableScan := FALSE;
END_IF

IF enableScan THEN
	// 输出一定长度的高电平;
	Welding_Arm_Digital_Outputs.16 := NOT ScanTon.Q;
	Digital_Outputs_16 := Welding_Arm_Digital_Outputs.16;
	Welding_Arm_Control.Axis_Relative_Eable[1] := FALSE;
ELSE
	Welding_Arm_Digital_Outputs.16 := 0;
END_IF

IF Trigger THEN
	IF LScanCounts < LScanRange/LScanStepSize THEN
		IF Welding_Arm_Control.MoveRelativeDone[1] THEN
			LScanCounts := LScanCounts + 1;
		END_IF		
	END_IF
ELSE
	Welding_Arm_Digital_Outputs :=0;
END_IF

IF LScanCounts >= LScanRange/LScanStepSize THEN
	Trigger :=0;
	LScanCounts := 0;
END_IF
END_ACTION

ACTION Signal_Monitor:

END_ACTION

END_PROGRAM

// ---- GlobalTextList.TcGTLO
TEXTLIST GlobalTextList
  145 = ' %.2f'
  240 = ' alpha_Terminal=%.3f'
  175 = ' realState=%.3f'
  165 = ' t_Interval=%.2f'
  167 = ' t_Interval=%.3f'
  169 = ' t_Interval=%.4f'
  168 = ' t_Interval=%.5f'
  300 = ' V = %.3f'
  241 = ' V=%.3f'
  297 = ' Xt = %.3f'
  244 = ' X_Act=%.3f'
  339 = ' X_t = %.3f'
  239 = ' X_Terminal=%.3f'
  245 = ' Y_Act=%.3f'
  325 = ' Zt = %.3'
  298 = ' Zt = %.3f'
  323 = ' Zt = %.3fm'
  324 = ' Zt = %.3m'
  296 = ' Zt=%.3f'
  243 = ' Z_Act=%.3f'
  238 = ' Z_Terminal=%.3f'
  143 = '%.2f'
  265 = '%.2f mm/s'
  217 = '%.3f'
  264 = '%.4f mm'
  207 = '%.4f mm/s'
  206 = '%.6f mm'
  179 = '1'
  293 = '134/246腿找零完成状态'
  305 = '135腿'
  287 = '135腿找零'
  306 = '246腿'
  288 = '246腿找零'
  263 = 'ALL_ENABLE'
  236 = 'Arm_Home_Done'
  254 = 'Auto_Moving'
  81 = 'Axis10_Back'
  82 = 'Axis10_Home'
  117 = 'Axis10_Move'
  11 = 'Axis10_Power'
  83 = 'Axis11_Back'
  84 = 'Axis11_Home'
  118 = 'Axis11_Move'
  12 = 'Axis11_Power'
  85 = 'Axis12_Back'
  86 = 'Axis12_Home'
  119 = 'Axis12_Move'
  13 = 'Axis12_Power'
  87 = 'Axis13_Back'
  88 = 'Axis13_Home'
  120 = 'Axis13_Move'
  14 = 'Axis13_Power'
  89 = 'Axis14_Back'
  90 = 'Axis14_Home'
  121 = 'Axis14_Move'
  15 = 'Axis14_Power'
  91 = 'Axis15_Back'
  92 = 'Axis15_Home'
  122 = 'Axis15_Move'
  16 = 'Axis15_Power'
  93 = 'Axis16_Back'
  94 = 'Axis16_Home'
  123 = 'Axis16_Move'
  17 = 'Axis16_Power'
  95 = 'Axis17_Back'
  96 = 'Axis17_Home'
  124 = 'Axis17_Move'
  18 = 'Axis17_Power'
  97 = 'Axis18_Back'
  98 = 'Axis18_Home'
  125 = 'Axis18_Move'
  19 = 'Axis18_Power'
  62 = 'Axis1_Back'
  64 = 'Axis1_Home'
  63 = 'Axis1_Home_Set'
  106 = 'Axis1_M'
  108 = 'Axis1_Move'
  2 = 'Axis1_Power'
  65 = 'Axis2_Back'
  66 = 'Axis2_Home'
  109 = 'Axis2_Move'
  3 = 'Axis2_Power'
  67 = 'Axis3_Back'
  68 = 'Axis3_Home'
  110 = 'Axis3_Move'
  4 = 'Axis3_Power'
  69 = 'Axis4_Back'
  70 = 'Axis4_Home'
  111 = 'Axis4_Move'
  5 = 'Axis4_Power'
  71 = 'Axis5_Back'
  72 = 'Axis5_Home'
  112 = 'Axis5_Move'
  6 = 'Axis5_Power'
  73 = 'Axis6_Back'
  74 = 'Axis6_Home'
  113 = 'Axis6_Move'
  7 = 'Axis6_Power'
  75 = 'Axis7_Back'
  76 = 'Axis7_Home'
  114 = 'Axis7_Move'
  8 = 'Axis7_Power'
  77 = 'Axis8_Back'
  78 = 'Axis8_Home'
  115 = 'Axis8_Move'
  9 = 'Axis8_Power'
  79 = 'Axis9_Back'
  80 = 'Axis9_Home'
  116 = 'Axis9_Move'
  10 = 'Axis9_Power'
  56 = 'Axis_ActPostion[INDEX]'
  60 = 'Back'
  174 = 'Botton For Step'
  309 = 'CoM(质心)实际位置'
  246 = 'CoM_Act'
  308 = 'CoM实际位置'
  334 = 'CoM（质心）实际位置'
  57 = 'Current_Turque_Value[INDEX]'
  211 = 'Drive1_Reset'
  212 = 'Drive2_Reset'
  213 = 'Drive3_Reset'
  214 = 'Drive4_Reset'
  215 = 'Drive5_Reset'
  216 = 'Drive6_Reset'
  39 = 'Driver10_Reset'
  40 = 'Driver11_Reset'
  41 = 'Driver12_Reset'
  42 = 'Driver13_Reset'
  43 = 'Driver14_Reset'
  44 = 'Driver15_Reset'
  45 = 'Driver16_Reset'
  46 = 'Driver17_Reset'
  47 = 'Driver18_Reset'
  30 = 'Driver1_Reset'
  31 = 'Driver2_Reset'
  32 = 'Driver3_Reset'
  33 = 'Driver4_Reset'
  34 = 'Driver5_Reset'
  35 = 'Driver6_Reset'
  36 = 'Driver7_Reset'
  37 = 'Driver8_Reset'
  38 = 'Driver9_Reset'
  341 = 'Enable_All_Buttons'
  313 = 'Enable_All_Units'
  274 = 'Enable_Overall_Units'
  209 = 'Error'
  127 = 'Error & Reset'
  126 = 'Error&Reset'
  151 = 'Exsetopint_Enable'
  152 = 'Exsetopint_On'
  141 = 'Exsetpoint_Exectue'
  23 = 'Home'
  230 = 'Home_Dont'
  231 = 'Home_DRobot_Home_Done'
  59 = 'Home_Execute'
  61 = 'Home_Set'
  227 = 'Leg135_Home'
  131 = 'Leg1_Home'
  181 = 'Leg21'
  228 = 'Leg246_Home'
  132 = 'Leg2_Home'
  133 = 'Leg3_Home'
  134 = 'Leg4_Home'
  135 = 'Leg5_Home'
  136 = 'Leg6_Home'
  180 = 'Leg_1'
  186 = 'Leg_16'
  182 = 'Leg_2'
  183 = 'Leg_3'
  184 = 'Leg_4'
  185 = 'Leg_5'
  187 = 'Leg_6'
  342 = 'Leg_Home_Done'
  177 = 'Model_Position[INDEX]'
  261 = 'Move'
  130 = 'Move & Stand'
  107 = 'MoveAbsoluteDone[INDEX]'
  129 = 'Move_Execute'
  223 = 'On'
  53 = 'Power'
  20 = 'Power_Execute'
  226 = 'Power_On'
  188 = 'RealState=%.3f'
  29 = 'Reset'
  49 = 'Reset_Execute'
  247 = 'Robot_Action'
  26 = 'Robot_Error'
  232 = 'Robot_Home_Done'
  101 = 'Robot_Home_Set'
  0 = 'Robot_Power'
  48 = 'Robot_Reset'
  128 = 'Robot_Stand_Execute'
  99 = 'Robot_Start_Back'
  100 = 'sadad'
  166 = 'Simulink_Move'
  270 = 'Simulink控制区域'
  176 = 'State=%.3f'
  189 = 'Step_Test'
  147 = 't=%.2f'
  170 = 't=%.3f'
  171 = 'Touch_Signal'
  178 = 'Touch_Signal(模型中腿编号)'
  172 = 'Touch_Signal_1'
  173 = 'Touch_Signal_Change'
  144 = 'T_ALL = %.2f'
  158 = 't_Interval=%.2f'
  242 = 'User_Control'
  248 = 'Walking_Robot'
  281 = 'Walking_Robot_Error'
  280 = 'Walking_Robot_Power'
  249 = 'Welding_Arm'
  235 = 'Welding_ArmHome_Done'
  194 = 'Welding_Arm_Error'
  229 = 'Welding_Arm_Home'
  234 = 'Welding_Arm_Home_Done'
  195 = 'Welding_Arm_Power'
  233 = 'Welding_Arnt_Home_Done'
  299 = 'αt = %.3f'
  191 = '上电操作'
  266 = '上电操作区域'
  250 = '信号监测'
  273 = '停止运动信号:'
  272 = '停止运动终止信号:'
  316 = '六足'
  336 = '六足、运动'
  318 = '六足上电'
  282 = '六足上电状态'
  317 = '六足坐标系示意图'
  315 = '六足机器人坐标示意图'
  335 = '六足正在运动'
  311 = '六足运动'
  319 = '六足错误'
  283 = '六足错误状态'
  284 = '关键状态监测'
  22 = '切换视图'
  157 = '取样时间间隔 t_Interval'
  160 = '取样时间间隔 t_Interval(ms)'
  161 = '取样时间间隔 t_Interval(s)'
  159 = '取样时间间隔 t_Interval/ms'
  220 = '取样间隔 t_Interval(s):'
  139 = '可以用来整体机器人运动'
  140 = '可以用来整体机器人进行Simulink模型验证'
  104 = '可以用来给单个四缸伸长或者是整体机器人站立'
  28 = '可以用来给单个电机或者是整体机器人上电'
  55 = '可以用来给单个电机或者是整体机器人找零'
  103 = '可以用来给单个电机或者是整体机器人站立'
  52 = '可以用来错误时给单个电机或者是整体机器人进行驱动重置'
  24 = '否'
  197 = '复位操作'
  292 = '对应找零完成状态'
  332 = '开始行走'
  333 = '开始行走到目标位置'
  338 = '开始行走至目标位置'
  222 = '开始输入目标运动轨迹'
  149 = '开始输入轨迹'
  301 = '开始运动信号'
  156 = '当前取样时间 t'
  163 = '当前取样时间 t(s)'
  218 = '当前取样时间 t(s):'
  295 = '找零完成状态'
  193 = '找零操作'
  268 = '找零操作区域'
  252 = '操作选择'
  255 = '整体移动焊接机器人控制系统'
  275 = '整体联合控制'
  25 = '是'
  204 = '是否允许找零操作'
  312 = '是否允许此界面操作'
  329 = '是否允许运动操作'
  203 = '是否允许通电操作'
  148 = '是否开始输入轨迹'
  328 = '是否激活此界面操作'
  198 = '是否进行Simulink运动操作'
  21 = '是否进行上电操作'
  303 = '是否进行子机找零'
  58 = '是否进行找零操作'
  302 = '是否进行整体上电'
  190 = '是否进行整机上电'
  192 = '是否进行整机找零'
  1 = '是否进行整机操作'
  142 = '是否进行运动操作'
  50 = '是否进行驱动重置'
  322 = '暂时没有'
  199 = '本界面为Welding-Arm操作界面'
  276 = '本界面为整体移动焊接机器人操作界面'
  225 = '本界面为整体移动焊接机器人操作界面：'
  138 = '本界面为电机Sumulink模型运动程序：'
  137 = '本界面为电机Sumulink程序：'
  27 = '本界面为电机上电程序：'
  102 = '本界面为电机伸长/机器人站立程序：'
  54 = '本界面为电机找零程序：'
  105 = '本界面为电机绝对运动/机器人站立程序：'
  201 = '本界面为移动焊机机器人联合控制界面'
  51 = '本界面为驱动重置程序：'
  202 = '本界面用于焊接臂上电及找零操作'
  269 = '本界面用于焊接臂运动及控制操作'
  208 = '本界面用于焊接臂运动控制操作'
  251 = '机器人坐标系示意'
  258 = '步行机器人调试与控制'
  260 = '步行移动焊接机器人控制系统'
  307 = '焊接臂'
  289 = '焊接臂6电机找零'
  320 = '焊接臂上电'
  285 = '焊接臂上电状态'
  304 = '焊接臂找零'
  294 = '焊接臂找零完成状态'
  259 = '焊接臂调试与控制'
  310 = '焊接臂运动'
  321 = '焊接臂错误'
  286 = '焊接臂错误状态'
  314 = '状态监测'
  267 = '状态监测区域'
  237 = '用户操作控制'
  291 = '用户自定义行走'
  278 = '用户自定义运动'
  277 = '用户自定义运动制'
  256 = '移动焊接机器人控制系统'
  257 = '联合控制'
  253 = '自主规划控制'
  331 = '自主规划行走'
  279 = '自主规划运动'
  330 = '自主规行走划运动'
  337 = '自主运动使能'
  290 = '行走开始'
  224 = '转到上电/找零'
  205 = '转到运动控制'
  154 = '输入运动总时长 T_ALL'
  162 = '输入运动总时长 T_ALL(s)'
  327 = '运动使能'
  262 = '运动开始'
  150 = '运动当前时间 t'
  164 = '运动当前时间 t(s)'
  146 = '运动总时长 T_ALL'
  196 = '运动总时长 T_ALL(s)'
  221 = '运动总时长 T_ALL(s):'
  200 = '运动操作'
  155 = '运动时间间隔 t'
  153 = '运动终止信号'
  219 = '运动终止信号:'
  326 = '运运动使能'
  340 = '这块还没完成'
  210 = '进行Simulink运动操作'
  271 = '驱动重设区域'
END_TEXTLIST

// ---- VISUs/Visu_Welding_Arm_Power.TcVIS
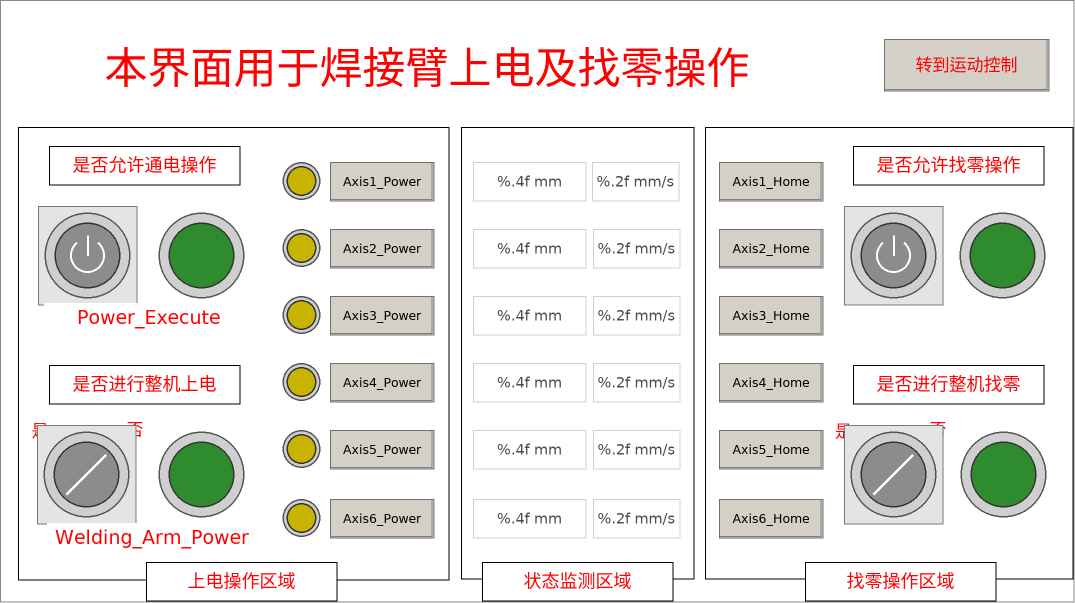
VISUALIZATION Visu_Welding_Arm_Power  // 1075x603
    Rectangle (705,127 368x452)
    Rectangle (461,127 233x452)
    Rectangle (18,127 431x453)
    Label (26,34 802x69), "本界面用于焊接臂上电及找零操作"
    Label (10,416 60x30), "是"
    RoundedRectangle (49,365 191x39), "是否进行整机上电"
    Label (108,416 54x27), "否"
    RoundedRectangle (49,146 191x39), "是否允许通电操作"
    Lamp1 (152,205 99x101), variable: Welding_Arm_Control.Power_Execute, style: Lamp-Lamp1-Green
    PowerSwitch (38,205 99x101), variable: Welding_Arm_Control.Power_Execute, behaviour: TOGGLE, style: Switch-PowerSwitch-Gray
    Lamp1 (152,424 99x101), variable: Welding_Arm_Control.Welding_Arm_Power, style: Lamp-Lamp1-Green
    RotarySwitch (37,424 99x101), variable: Welding_Arm_Control.Welding_Arm_Power, behaviour: TOGGLE, style: Switch-RotarySwitch-Gray
    Label (812,417 63x29), "是"
    RoundedRectangle (853,365 191x39), "是否进行整机找零"
    Label (911,416 54x27), "否"
    RoundedRectangle (853,146 191x39), "是否允许找零操作"
    Lamp1 (953,205 99x101), variable: Welding_Arm_Control.Home_Execute, style: Lamp-Lamp1-Green
    PowerSwitch (844,205 99x101), variable: Welding_Arm_Control.Home_Execute, behaviour: TOGGLE, style: Switch-PowerSwitch-Gray
    Lamp1 (954,424 99x101), variable: Welding_Arm_Control.Welding_Arm_Home_Set, style: Lamp-Lamp1-Green
    RotarySwitch (844,424 99x101), variable: Welding_Arm_Control.Welding_Arm_Home_Set, behaviour: TOGGLE, style: Switch-RotarySwitch-Gray
    Button (884,39 165x52), "转到运动控制"
        OnMouseClick: change screen: Visu_Welding_Arm_SimulinkMove
    Lamp1 (274,159 55x44), variable: Welding_Arm_Control.Power_Status[1], style: Lamp-Lamp1-Yellow
    Button (330,162 104x39), "Axis1_Power"
        toggle Welding_Arm_Control.Axis_Power[1]
    Button (719,162 104x39), "Axis1_Home"
        toggle Welding_Arm_Control.Axis_Home_Set[1]
    Textfield (473,162 113x39), "%.4f mm", text variable: Welding_Arm_Control.Axis_ActPostion[1]
    Textfield (592,162 87x39), "%.2f mm/s", text variable: Welding_Arm_Control.Axis_ActVelocity[1]
    Lamp1 (274,226 55x44), variable: Welding_Arm_Control.Power_Status[2], style: Lamp-Lamp1-Yellow
    Button (330,229 104x39), "Axis2_Power"
        toggle Welding_Arm_Control.Axis_Power[2]
    Button (719,229 104x39), "Axis2_Home"
        toggle Welding_Arm_Control.Axis_Home_Set[2]
    Textfield (473,229 113x39), "%.4f mm", text variable: Welding_Arm_Control.Axis_ActPostion[2]
    Textfield (593,229 87x39), "%.2f mm/s", text variable: Welding_Arm_Control.Axis_ActVelocity[2]
    Lamp1 (274,293 55x44), variable: Welding_Arm_Control.Power_Status[3], style: Lamp-Lamp1-Yellow
    Button (330,296 104x39), "Axis3_Power"
        toggle Welding_Arm_Control.Axis_Power[3]
    Button (719,296 104x39), "Axis3_Home"
        toggle Welding_Arm_Control.Axis_Home_Set[3]
    Textfield (473,296 113x39), "%.4f mm", text variable: Welding_Arm_Control.Axis_ActPostion[3]
    Textfield (593,296 87x39), "%.2f mm/s", text variable: Welding_Arm_Control.Axis_ActVelocity[3]
    Lamp1 (274,360 55x44), variable: Welding_Arm_Control.Power_Status[4], style: Lamp-Lamp1-Yellow
    Button (330,363 104x39), "Axis4_Power"
        toggle Welding_Arm_Control.Axis_Power[4]
    Button (719,363 104x39), "Axis4_Home"
        toggle Welding_Arm_Control.Axis_Home_Set[4]
    Textfield (473,363 113x39), "%.4f mm", text variable: Welding_Arm_Control.Axis_ActPostion[4]
    Textfield (593,363 87x39), "%.2f mm/s", text variable: Welding_Arm_Control.Axis_ActVelocity[4]
    Lamp1 (274,427 55x44), variable: Welding_Arm_Control.Power_Status[5], style: Lamp-Lamp1-Yellow
    Button (330,430 104x39), "Axis5_Power"
        toggle Welding_Arm_Control.Axis_Power[5]
    Button (719,430 104x39), "Axis5_Home"
        toggle Welding_Arm_Control.Axis_Home_Set[5]
    Textfield (473,430 113x39), "%.4f mm", text variable: Welding_Arm_Control.Axis_ActPostion[5]
    Textfield (593,430 87x39), "%.2f mm/s", text variable: Welding_Arm_Control.Axis_ActVelocity[5]
    Lamp1 (274,496 55x44), variable: Welding_Arm_Control.Power_Status[6], style: Lamp-Lamp1-Yellow
    Button (330,499 104x39), "Axis6_Power"
        toggle Welding_Arm_Control.Axis_Power[6]
    Button (719,499 104x39), "Axis6_Home"
        toggle Welding_Arm_Control.Axis_Home_Set[6]
    Textfield (473,499 113x39), "%.4f mm", text variable: Welding_Arm_Control.Axis_ActPostion[6]
    Textfield (593,499 87x39), "%.2f mm/s", text variable: Welding_Arm_Control.Axis_ActVelocity[6]
    RoundedRectangle (146,562 191x39), "上电操作区域"
    RoundedRectangle (482,562 191x39), "状态监测区域"
    Rectangle (44,303 210x29), "Power_Execute"
    Rectangle (47,523 210x29), "Welding_Arm_Power"
    RoundedRectangle (805,562 191x39), "找零操作区域"
END_VISUALIZATION

// ---- VISUs/Visu_Welding_Arm_SimulinkMove.TcVIS
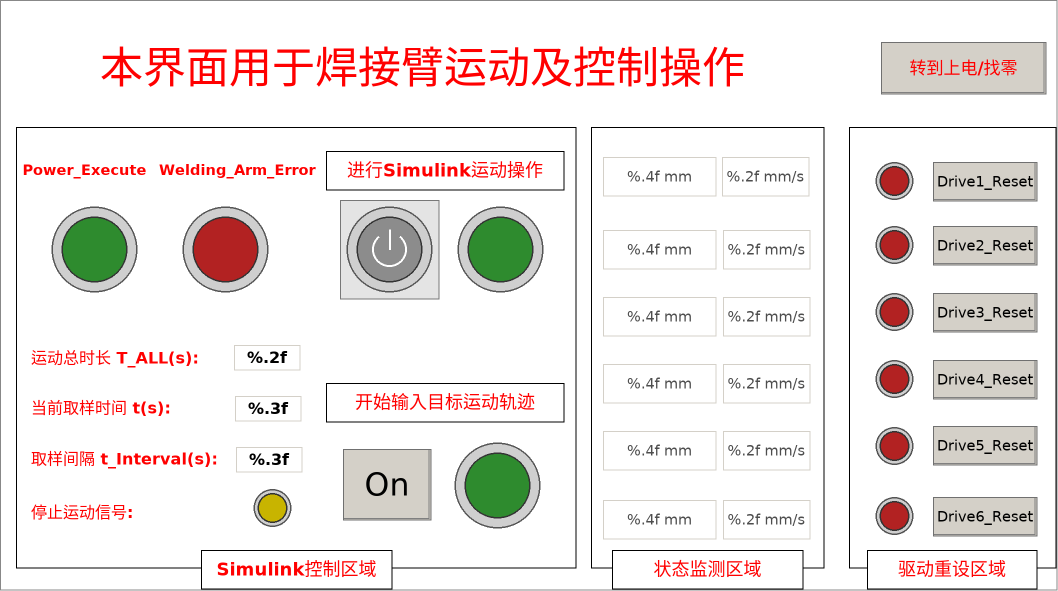
VISUALIZATION Visu_Welding_Arm_SimulinkMove  // 1058x591
    Rectangle (849,127 207x441)
    Rectangle (16,127 560x441)
    Label (19,154 131x32), "Power_Execute"
    Label (160,154 155x32), "Welding_Arm_Error"
    RoundedRectangle (326,151 238x39), "进行Simulink运动操作"
    Lamp1 (451,199 99x101), variable: Welding_Arm_Movement.ExSetPoint_Execute, style: Lamp-Lamp1-Green
    PowerSwitch (340,199 99x101), variable: Welding_Arm_Movement.ExSetPoint_Execute, behaviour: TOGGLE, style: Switch-PowerSwitch-Gray
    Lamp1 (867,159 55x44), variable: Welding_Arm_Control.Axis_Error[1], style: Lamp-Lamp1-Red
    Button (933,162 104x39), "Drive1_Reset"
        toggle Welding_Arm_Control.Axis_Reset[1]
    Lamp1 (867,223 55x44), variable: Welding_Arm_Control.Axis_Error[2], style: Lamp-Lamp1-Red
    Button (933,226 104x39), "Drive2_Reset"
        toggle Welding_Arm_Control.Axis_Reset[2]
    Lamp1 (867,290 55x44), variable: Welding_Arm_Control.Axis_Error[3], style: Lamp-Lamp1-Red
    Button (933,293 104x39), "Drive3_Reset"
        toggle Welding_Arm_Control.Axis_Reset[3]
    Lamp1 (867,357 55x44), variable: Welding_Arm_Control.Axis_Error[4], style: Lamp-Lamp1-Red
    Button (933,360 104x39), "Drive4_Reset"
        toggle Welding_Arm_Control.Axis_Reset[4]
    Lamp1 (867,424 55x44), variable: Welding_Arm_Control.Axis_Error[5], style: Lamp-Lamp1-Red
    Button (933,426 104x39), "Drive5_Reset"
        toggle Welding_Arm_Control.Axis_Reset[5]
    Lamp1 (867,494 55x44), variable: Welding_Arm_Control.Axis_Error[6], style: Lamp-Lamp1-Red
    Button (933,497 104x39), "Drive6_Reset"
        toggle Welding_Arm_Control.Axis_Reset[6]
    Textfield (235,396 66x25), "%.3f", text variable: Welding_Arm_Movement.t
    Label (28,396 188x24), "当前取样时间 t(s):"
    Lamp1 (245,486 55x44), variable: Welding_Arm_Movement.ExtSetPointDisable, style: Lamp-Lamp1-Yellow
    Label (28,499 182x27), "停止运动信号:"
    Label (28,447 205x24), "取样间隔 t_Interval(s):"
    Textfield (236,447 66x25), "%.3f", text variable: Welding_Arm_Movement.t_Interval
        OnMouseClick: write Welding_Arm_Movement.t_Interval via Default
    Label (28,346 199x24), "运动总时长 T_ALL(s):"
    Textfield (234,345 66x25), "%.2f", text variable: Welding_Arm_Movement.T_ALL
    RoundedRectangle (326,383 238x39), "开始输入目标运动轨迹"
    Lamp1 (448,435 99x101), variable: Welding_Arm_Movement.ExtSetPointEnable, style: Lamp-Lamp1-Green
    Button (343,449 88x71), "On"
        toggle Welding_Arm_Movement.ExtSetPointEnable
    Button (881,42 165x52), "转到上电/找零"
        OnMouseClick: change screen: Visu_Welding_Arm_Power
    Lamp1 (176,199 99x101), variable: Welding_Arm_Control.Welding_Arm_Error, style: Lamp-Lamp1-Red
    Lamp1 (45,199 99x101), variable: Welding_Arm_Control.Power_Execute, style: Lamp-Lamp1-Green
    Label (16,38 813x60), "本界面用于焊接臂运动及控制操作"
    RoundedRectangle (201,550 191x39), "Simulink控制区域"
    Rectangle (591,127 233x441)
    Textfield (603,157 113x39), "%.4f mm", text variable: Welding_Arm_Control.Axis_ActPostion[1]
    Textfield (722,157 87x39), "%.2f mm/s", text variable: Welding_Arm_Control.Axis_ActVelocity[1]
    Textfield (603,230 113x39), "%.4f mm", text variable: Welding_Arm_Control.Axis_ActPostion[2]
    Textfield (723,230 87x39), "%.2f mm/s", text variable: Welding_Arm_Control.Axis_ActVelocity[2]
    Textfield (603,297 113x39), "%.4f mm", text variable: Welding_Arm_Control.Axis_ActPostion[3]
    Textfield (723,297 87x39), "%.2f mm/s", text variable: Welding_Arm_Control.Axis_ActVelocity[3]
    Textfield (603,364 113x39), "%.4f mm", text variable: Welding_Arm_Control.Axis_ActPostion[4]
    Textfield (723,364 87x39), "%.2f mm/s", text variable: Welding_Arm_Control.Axis_ActVelocity[4]
    Textfield (603,431 113x39), "%.4f mm", text variable: Welding_Arm_Control.Axis_ActPostion[5]
    Textfield (723,431 87x39), "%.2f mm/s", text variable: Welding_Arm_Control.Axis_ActVelocity[5]
    Textfield (603,500 113x39), "%.4f mm", text variable: Welding_Arm_Control.Axis_ActPostion[6]
    Textfield (723,500 87x39), "%.2f mm/s", text variable: Welding_Arm_Control.Axis_ActVelocity[6]
    RoundedRectangle (612,550 191x39), "状态监测区域"
    RoundedRectangle (867,550 170x39), "驱动重设区域"
END_VISUALIZATION

// ---- VISUs/Visu_Walking_Robot_Home.TcVIS
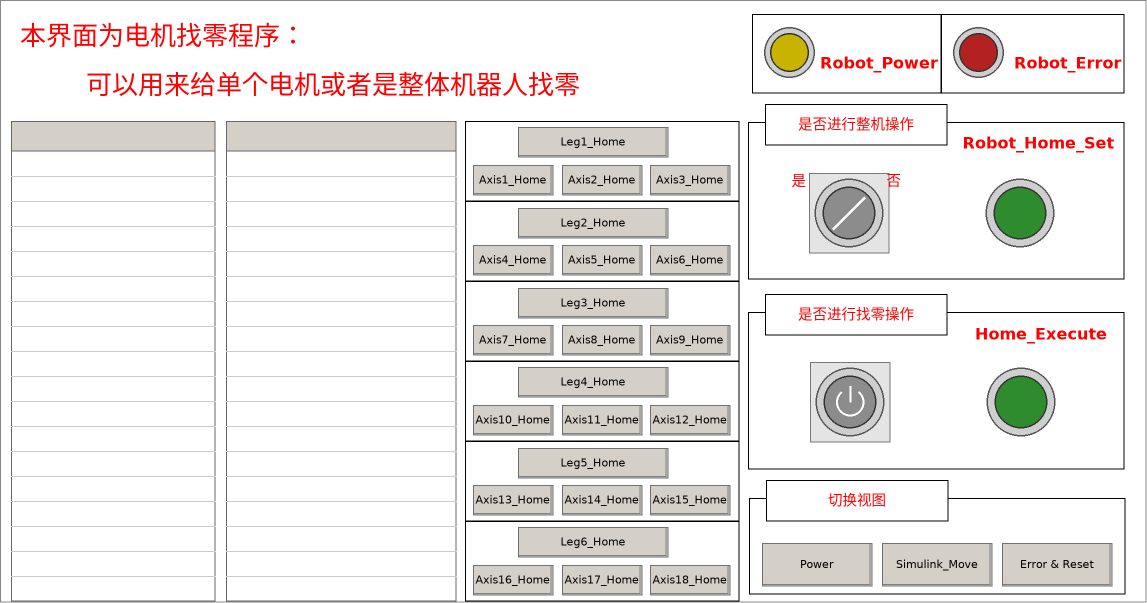
VISUALIZATION Visu_Walking_Robot_Home  // 1147x603
    Rectangle (752,14 189x79)
    Rectangle (748,312 376x157)
    Label (964,318 154x32), "Home_Execute"
    Rectangle (765,294 182x41), "是否进行找零操作"
    Lamp1 (981,362 80x80), variable: Walking_Robot_Control.Home_Execute, style: Lamp-Lamp1-Green
    PowerSwitch (810,362 80x80), variable: Walking_Robot_Control.Home_Execute, behaviour: TOGGLE, style: Switch-PowerSwitch-Gray
    Rectangle (941,14 183x79)
    Lamp1 (948,23 61x59), variable: Walking_Robot_Control.Robot_Error, style: Lamp-Lamp1-Red
    Label (991,47 154x32), "Robot_Error"
    Label (17,15 365x42), "本界面为电机找零程序："
    Label (83,64 874x42), "可以用来给单个电机或者是整体机器人找零"
    Table (11,121 204x480), data array: Walking_Robot_Control.Axis_ActPostion
        p3854506369: Walking_Robot_Control.Axis_ActPostion[INDEX]
    Table (226,121 230x480), data array: Walking_Robot_Control.Current_Turque_Value
        p3854506369: Walking_Robot_Control.Current_Turque_Value[INDEX]
    Lamp1 (759,23 61x59), variable: Walking_Robot_Control.Robot_Power, style: Lamp-Lamp1-Yellow
    Label (802,47 154x32), "Robot_Power"
    Rectangle (465,121 274x80)
    Button (473,165 80x30), "Axis1_Home"
        toggle Walking_Robot_Control.Axis_Home_Set[1]
        OnMouseClick: change screen: Visu_Home
    Button (650,165 80x30), "Axis3_Home"
        toggle Walking_Robot_Control.Axis_Home_Set[3]
        OnMouseClick: change screen: Visu_Home
    Button (562,165 80x30), "Axis2_Home"
        toggle Walking_Robot_Control.Axis_Home_Set[2]
        OnMouseClick: change screen: Visu_Home
    Rectangle (465,201 274x80)
    Button (473,245 80x30), "Axis4_Home"
        toggle Walking_Robot_Control.Axis_Home_Set[4]
        OnMouseClick: change screen: Visu_Home
    Button (650,245 80x30), "Axis6_Home"
        toggle Walking_Robot_Control.Axis_Home_Set[6]
        OnMouseClick: change screen: Visu_Home
    Button (562,245 80x30), "Axis5_Home"
        toggle Walking_Robot_Control.Axis_Home_Set[5]
        OnMouseClick: change screen: Visu_Home
    Rectangle (465,281 274x80)
    Button (473,325 80x30), "Axis7_Home"
        toggle Walking_Robot_Control.Axis_Home_Set[7]
        OnMouseClick: change screen: Visu_Home
    Button (650,325 80x30), "Axis9_Home"
        toggle Walking_Robot_Control.Axis_Home_Set[9]
        OnMouseClick: change screen: Visu_Home
    Button (562,325 80x30), "Axis8_Home"
        toggle Walking_Robot_Control.Axis_Home_Set[8]
        OnMouseClick: change screen: Visu_Home
    Rectangle (465,361 274x80)
    Button (473,405 80x30), "Axis10_Home"
        toggle Walking_Robot_Control.Axis_Home_Set[10]
        OnMouseClick: change screen: Visu_Home
    Button (650,405 80x30), "Axis12_Home"
        toggle Walking_Robot_Control.Axis_Home_Set[12]
        OnMouseClick: change screen: Visu_Home
    Button (562,405 80x30), "Axis11_Home"
        toggle Walking_Robot_Control.Axis_Home_Set[11]
        OnMouseClick: change screen: Visu_Home
    Rectangle (465,441 274x80)
    Button (473,485 80x30), "Axis13_Home"
        toggle Walking_Robot_Control.Axis_Home_Set[13]
        OnMouseClick: change screen: Visu_Home
    Button (650,485 80x30), "Axis15_Home"
        toggle Walking_Robot_Control.Axis_Home_Set[15]
        OnMouseClick: change screen: Visu_Home
    Button (562,485 80x30), "Axis14_Home"
        toggle Walking_Robot_Control.Axis_Home_Set[14]
        OnMouseClick: change screen: Visu_Home
    Rectangle (465,521 274x80)
    Button (473,565 80x30), "Axis16_Home"
        toggle Walking_Robot_Control.Axis_Home_Set[16]
        OnMouseClick: change screen: Visu_Home
    Button (650,565 80x30), "Axis18_Home"
        toggle Walking_Robot_Control.Axis_Home_Set[18]
        OnMouseClick: change screen: Visu_Home
    Button (562,565 80x30), "Axis17_Home"
        toggle Walking_Robot_Control.Axis_Home_Set[17]
        OnMouseClick: change screen: Visu_Home
    Rectangle (749,498 376x96)
    Rectangle (766,480 182x41), "切换视图"
    Button (762,543 110x43), "Power"
        OnMouseClick: change screen: Visu_Walking_Robot_Power
    Button (1002,543 110x43), "Error & Reset"
        OnMouseClick: change screen: Visu_Walking_Robot_Reset
    Button (882,543 110x43), "Simulink_Move"
        OnMouseClick: change screen: Visu_Walking_Robot_SimulinkMove
    Rectangle (748,122 376x157)
    Rectangle (765,104 182x41), "是否进行整机操作"
    Lamp1 (980,173 80x80), variable: Walking_Robot_Control.Robot_Home_Set, style: Lamp-Lamp1-Green
    RotarySwitch (809,173 80x80), variable: Walking_Robot_Control.Robot_Home_Set, behaviour: TOGGLE, style: Switch-RotarySwitch-Gray
    Label (864,166 60x30), "否"
    Label (769,166 60x30), "是"
    Label (935,127 207x32), "Robot_Home_Set"
    Button (518,127 150x30), "Leg1_Home"
        tap Walking_Robot_Control.Leg_Home_Set[1]
    Button (518,208 150x30), "Leg2_Home"
        tap Walking_Robot_Control.Leg_Home_Set[2]
    Button (518,288 150x30), "Leg3_Home"
        tap Walking_Robot_Control.Leg_Home_Set[3]
    Button (518,367 150x30), "Leg4_Home"
        tap Walking_Robot_Control.Leg_Home_Set[4]
    Button (518,448 150x30), "Leg5_Home"
        tap Walking_Robot_Control.Leg_Home_Set[5]
    Button (518,527 150x30), "Leg6_Home"
        tap Walking_Robot_Control.Leg_Home_Set[6]
END_VISUALIZATION

// ---- VISUs/Visu_Walking_Robot_Power.TcVIS
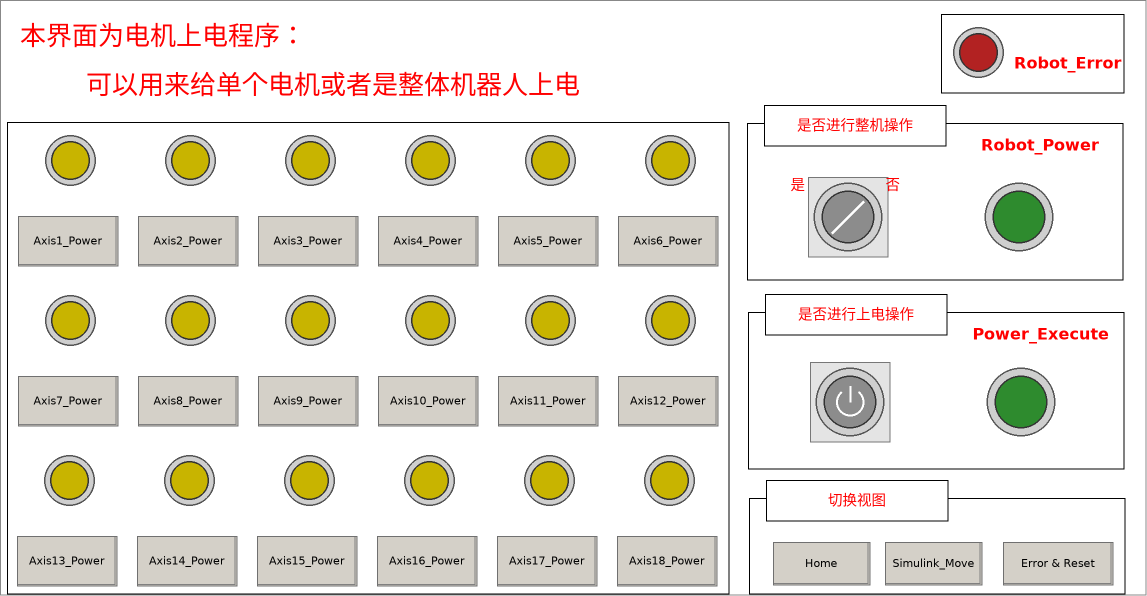
VISUALIZATION Visu_Walking_Robot_Power  // 1147x596
    Label (987,37 154x32), "Robot_Error"
    Rectangle (7,122 722x472)
    Lamp1 (40,131 61x59), variable: Walking_Robot_Control.Power_Status[1], style: Lamp-Lamp1-Yellow
    Lamp1 (160,131 61x59), variable: Walking_Robot_Control.Power_Status[2], style: Lamp-Lamp1-Yellow
    Lamp1 (280,131 61x59), variable: Walking_Robot_Control.Power_Status[3], style: Lamp-Lamp1-Yellow
    Lamp1 (400,131 61x59), variable: Walking_Robot_Control.Power_Status[4], style: Lamp-Lamp1-Yellow
    Lamp1 (520,131 61x59), variable: Walking_Robot_Control.Power_Status[5], style: Lamp-Lamp1-Yellow
    Lamp1 (640,131 61x59), variable: Walking_Robot_Control.Power_Status[6], style: Lamp-Lamp1-Yellow
    Button (18,216 100x50), "Axis1_Power"
        toggle Walking_Robot_Control.Axis_Power[1]
    Button (138,216 100x50), "Axis2_Power"
        toggle Walking_Robot_Control.Axis_Power[2]
    Button (258,216 100x50), "Axis3_Power"
        toggle Walking_Robot_Control.Axis_Power[3]
    Button (378,216 100x50), "Axis4_Power"
        toggle Walking_Robot_Control.Axis_Power[4]
    Button (498,216 100x50), "Axis5_Power"
        toggle Walking_Robot_Control.Axis_Power[5]
    Button (618,216 100x50), "Axis6_Power"
        toggle Walking_Robot_Control.Axis_Power[6]
    Lamp1 (40,291 61x59), variable: Walking_Robot_Control.Power_Status[7], style: Lamp-Lamp1-Yellow
    Lamp1 (160,291 61x59), variable: Walking_Robot_Control.Power_Status[8], style: Lamp-Lamp1-Yellow
    Lamp1 (280,291 61x59), variable: Walking_Robot_Control.Power_Status[9], style: Lamp-Lamp1-Yellow
    Lamp1 (400,291 61x59), variable: Walking_Robot_Control.Power_Status[10], style: Lamp-Lamp1-Yellow
    Lamp1 (520,291 61x59), variable: Walking_Robot_Control.Power_Status[11], style: Lamp-Lamp1-Yellow
    Lamp1 (640,291 61x59), variable: Walking_Robot_Control.Power_Status[12], style: Lamp-Lamp1-Yellow
    Button (18,376 100x50), "Axis7_Power"
        toggle Walking_Robot_Control.Axis_Power[7]
    Button (138,376 100x50), "Axis8_Power"
        toggle Walking_Robot_Control.Axis_Power[8]
    Button (258,376 100x50), "Axis9_Power"
        toggle Walking_Robot_Control.Axis_Power[9]
    Button (378,376 100x50), "Axis10_Power"
        toggle Walking_Robot_Control.Axis_Power[10]
    Button (498,376 100x50), "Axis11_Power"
        toggle Walking_Robot_Control.Axis_Power[11]
    Button (618,376 100x50), "Axis12_Power"
        toggle Walking_Robot_Control.Axis_Power[12]
    Lamp1 (39,451 61x59), variable: Walking_Robot_Control.Power_Status[13], style: Lamp-Lamp1-Yellow
    Lamp1 (159,451 61x59), variable: Walking_Robot_Control.Power_Status[14], style: Lamp-Lamp1-Yellow
    Lamp1 (279,451 61x59), variable: Walking_Robot_Control.Power_Status[15], style: Lamp-Lamp1-Yellow
    Lamp1 (399,451 61x59), variable: Walking_Robot_Control.Power_Status[16], style: Lamp-Lamp1-Yellow
    Lamp1 (519,451 61x59), variable: Walking_Robot_Control.Power_Status[17], style: Lamp-Lamp1-Yellow
    Lamp1 (639,451 61x59), variable: Walking_Robot_Control.Power_Status[18], style: Lamp-Lamp1-Yellow
    Button (17,536 100x50), "Axis13_Power"
        toggle Walking_Robot_Control.Axis_Power[13]
    Button (137,536 100x50), "Axis14_Power"
        toggle Walking_Robot_Control.Axis_Power[14]
    Button (257,536 100x50), "Axis15_Power"
        toggle Walking_Robot_Control.Axis_Power[15]
    Button (377,536 100x50), "Axis16_Power"
        toggle Walking_Robot_Control.Axis_Power[16]
    Button (497,536 100x50), "Axis17_Power"
        toggle Walking_Robot_Control.Axis_Power[17]
    Button (617,536 100x50), "Axis18_Power"
        toggle Walking_Robot_Control.Axis_Power[18]
    Rectangle (748,312 376x157)
    Label (964,318 154x32), "Power_Execute"
    Rectangle (765,294 182x41), "是否进行上电操作"
    Lamp1 (981,362 80x80), variable: Walking_Robot_Control.Power_Execute, style: Lamp-Lamp1-Green
    Rectangle (749,498 376x96)
    Rectangle (766,480 182x41), "切换视图"
    Button (773,542 97x43), "Home"
        OnMouseClick: change screen: Visu_Walking_Robot_Home
    PowerSwitch (810,362 80x80), variable: Walking_Robot_Control.Power_Execute, behaviour: TOGGLE, style: Switch-PowerSwitch-Gray
    Rectangle (941,14 183x79)
    Lamp1 (948,23 61x59), variable: Walking_Robot_Control.Robot_Error, style: Lamp-Lamp1-Red
    Label (17,15 365x42), "本界面为电机上电程序："
    Label (83,64 639x42), "可以用来给单个电机或者是整体机器人上电"
    Button (1003,542 110x43), "Error & Reset"
        OnMouseClick: change screen: Visu_Walking_Robot_Reset
    Rectangle (747,123 376x157)
    Label (963,129 154x32), "Robot_Power"
    Rectangle (764,105 182x41), "是否进行整机操作"
    Lamp1 (979,177 80x80), variable: Walking_Robot_Control.Robot_Power, style: Lamp-Lamp1-Green
    RotarySwitch (808,177 80x80), variable: Walking_Robot_Control.Robot_Power, behaviour: TOGGLE, style: Switch-RotarySwitch-Gray
    Label (863,170 60x30), "否"
    Label (768,170 60x30), "是"
    Label (991,47 154x32), "Robot_Error"
    Button (885,542 97x43), "Simulink_Move"
        OnMouseClick: change screen: Visu_Walking_Robot_SimulinkMove
END_VISUALIZATION

